LIN {X 99.483,Y -60.000,Z -86.142,A -90.000,B 90.000,C 0.000} C_DIS
LIN {X 99.483,Y -29.308,Z -86.142,A -90.000,B 90.000,C 0.000} C_DIS
LIN {X 99.474,Y -29.310,Z -86.271,A -90.000,B 90.000,C 0.000} C_DIS
LIN {X 99.431,Y -29.338,Z -86.823,A -90.000,B 90.000,C 0.000} C_DIS
LIN {X 99.416,Y -29.357,Z -87.009,A -90.000,B 90.000,C 0.000} C_DIS
LIN {X 99.411,Y -29.358,Z -87.066,A -90.000,B 90.000,C 0.000} C_DIS
LIN {X 99.408,Y -29.365,Z -87.238,A -90.000,B 90.000,C 0.000} C_DIS
LIN {X 99.404,Y -29.371,Z -87.535,A -90.000,B 90.000,C 0.000} C_DIS
LIN {X 99.396,Y -29.374,Z -87.741,A -90.000,B 90.000,C 0.000} C_DIS
LIN {X 99.366,Y -29.385,Z -88.382,A -90.000,B 90.000,C 0.000} C_DIS
LIN {X 99.349,Y -29.388,Z -88.757,A -90.000,B 90.000,C 0.000} C_DIS
LIN {X 99.326,Y -29.411,Z -90.340,A -90.000,B 90.000,C 0.000} C_DIS
LIN {X 99.319,Y -29.416,Z -90.874,A -90.000,B 90.000,C 0.000} C_DIS
LIN {X 99.295,Y -29.416,Z -91.496,A -90.000,B 90.000,C 0.000} C_DIS
LIN {X 99.271,Y -29.421,Z -92.100,A -90.000,B 90.000,C 0.000} C_DIS
LIN {X 99.242,Y -29.426,Z -92.749,A -90.000,B 90.000,C 0.000} C_DIS
LIN {X 99.174,Y -29.426,Z -93.750,A -90.000,B 90.000,C 0.000} C_DIS
LIN {X 99.148,Y -29.428,Z -94.121,A -90.000,B 90.000,C 0.000} C_DIS
LIN {X 99.143,Y -29.428,Z -94.158,A -90.000,B 90.000,C 0.000} C_DIS
LIN {X 99.082,Y -29.425,Z -94.592,A -90.000,B 90.000,C 0.000} C_DIS
LIN {X 98.973,Y -29.414,Z -95.189,A -90.000,B 90.000,C 0.000} C_DIS
LIN {X 98.893,Y -29.411,Z -95.613,A -90.000,B 90.000,C 0.000} C_DIS
LIN {X 98.843,Y -29.411,Z -95.835,A -90.000,B 90.000,C 0.000} C_DIS
LIN {X 98.623,Y -29.420,Z -96.806,A -90.000,B 90.000,C 0.000} C_DIS
LIN {X 98.597,Y -29.422,Z -96.941,A -90.000,B 90.000,C 0.000} C_DIS
LIN {X 98.549,Y -29.421,Z -97.133,A -90.000,B 90.000,C 0.000} C_DIS
LIN {X 98.489,Y -29.424,Z -97.369,A -90.000,B 90.000,C 0.000} C_DIS
LIN {X 98.242,Y -29.426,Z -98.215,A -90.000,B 90.000,C 0.000} C_DIS
LIN {X 98.196,Y -29.431,Z -98.439,A -90.000,B 90.000,C 0.000} C_DIS
LIN {X 98.116,Y -29.446,Z -98.815,A -90.000,B 90.000,C 0.000} C_DIS
LIN {X 98.030,Y -29.468,Z -99.250,A -90.000,B 90.000,C 0.000} C_DIS
LIN {X 97.907,Y -29.486,Z -99.897,A -90.000,B 90.000,C 0.000} C_DIS
LIN {X 97.776,Y -29.509,Z -100.630,A -90.000,B 90.000,C 0.000} C_DIS
LIN {X 97.672,Y -29.519,Z -101.231,A -90.000,B 90.000,C 0.000} C_DIS
LIN {X 97.614,Y -29.526,Z -101.574,A -90.000,B 90.000,C 0.000} C_DIS
LIN {X 97.555,Y -29.538,Z -101.977,A -90.000,B 90.000,C 0.000} C_DIS
LIN {X 97.524,Y -29.542,Z -102.200,A -90.000,B 90.000,C 0.000} C_DIS
LIN {X 97.389,Y -29.552,Z -103.092,A -90.000,B 90.000,C 0.000} C_DIS
LIN {X 97.380,Y -29.555,Z -103.178,A -90.000,B 90.000,C 0.000} C_DIS
LIN {X 97.349,Y -29.565,Z -103.442,A -90.000,B 90.000,C 0.000} C_DIS
LIN {X 97.261,Y -29.575,Z -104.227,A -90.000,B 90.000,C 0.000} C_DIS
LIN {X 97.256,Y -29.586,Z -104.403,A -90.000,B 90.000,C 0.000} C_DIS
LIN {X 97.253,Y -29.592,Z -104.507,A -90.000,B 90.000,C 0.000} C_DIS
LIN {X 97.252,Y -29.598,Z -105.008,A -90.000,B 90.000,C 0.000} C_DIS
LIN {X 97.255,Y -29.601,Z -105.049,A -90.000,B 90.000,C 0.000} C_DIS
LIN {X 97.332,Y -29.605,Z -105.759,A -90.000,B 90.000,C 0.000} C_DIS
LIN {X 97.345,Y -29.602,Z -105.867,A -90.000,B 90.000,C 0.000} C_DIS
LIN {X 97.415,Y -29.603,Z -106.286,A -90.000,B 90.000,C 0.000} C_DIS
LIN {X 97.518,Y -29.607,Z -106.935,A -90.000,B 90.000,C 0.000} C_DIS
LIN {X 97.664,Y -29.611,Z -107.964,A -90.000,B 90.000,C 0.000} C_DIS
LIN {X 97.689,Y -29.614,Z -108.147,A -90.000,B 90.000,C 0.000} C_DIS
LIN {X 97.799,Y -29.623,Z -109.641,A -90.000,B 90.000,C 0.000} C_DIS
LIN {X 97.823,Y -29.623,Z -110.079,A -90.000,B 90.000,C 0.000} C_DIS
LIN {X 97.850,Y -29.627,Z -110.772,A -90.000,B 90.000,C 0.000} C_DIS
LIN {X 97.887,Y -29.631,Z -111.828,A -90.000,B 90.000,C 0.000} C_DIS
LIN {X 97.974,Y -29.650,Z -115.821,A -90.000,B 90.000,C 0.000} C_DIS
LIN {X 98.033,Y -29.661,Z -117.860,A -90.000,B 90.000,C 0.000} C_DIS
LIN {X 98.103,Y -29.670,Z -120.291,A -90.000,B 90.000,C 0.000} C_DIS
LIN {X 98.151,Y -29.676,Z -122.571,A -90.000,B 90.000,C 0.000} C_DIS
LIN {X 98.155,Y -29.681,Z -124.129,A -90.000,B 90.000,C 0.000} C_DIS
LIN {X 98.155,Y -29.682,Z -124.889,A -90.000,B 90.000,C 0.000} C_DIS
LIN {X 98.140,Y -29.682,Z -125.406,A -90.000,B 90.000,C 0.000} C_DIS
LIN {X 98.088,Y -29.690,Z -127.201,A -90.000,B 90.000,C 0.000} C_DIS
LIN {X 98.040,Y -29.694,Z -128.030,A -90.000,B 90.000,C 0.000} C_DIS
LIN {X 97.964,Y -29.700,Z -129.451,A -90.000,B 90.000,C 0.000} C_DIS
LIN {X 97.879,Y -29.705,Z -130.608,A -90.000,B 90.000,C 0.000} C_DIS
LIN {X 97.791,Y -29.710,Z -131.863,A -90.000,B 90.000,C 0.000} C_DIS
LIN {X 97.673,Y -29.714,Z -133.353,A -90.000,B 90.000,C 0.000} C_DIS
LIN {X 97.534,Y -29.719,Z -135.178,A -90.000,B 90.000,C 0.000} C_DIS
LIN {X 97.341,Y -29.723,Z -137.704,A -90.000,B 90.000,C 0.000} C_DIS
LIN {X 97.283,Y -29.724,Z -138.417,A -90.000,B 90.000,C 0.000} C_DIS
LIN {X 97.044,Y -29.726,Z -141.288,A -90.000,B 90.000,C 0.000} C_DIS
LIN {X 97.013,Y -29.725,Z -141.637,A -90.000,B 90.000,C 0.000} C_DIS
LIN {X 96.932,Y -29.726,Z -142.492,A -90.000,B 90.000,C 0.000} C_DIS
LIN {X 96.735,Y -29.726,Z -144.533,A -90.000,B 90.000,C 0.000} C_DIS
LIN {X 96.664,Y -29.726,Z -145.241,A -90.000,B 90.000,C 0.000} C_DIS
LIN {X 96.504,Y -29.729,Z -146.660,A -90.000,B 90.000,C 0.000} C_DIS
LIN {X 96.220,Y -29.731,Z -149.069,A -90.000,B 90.000,C 0.000} C_DIS
LIN {X 96.032,Y -29.735,Z -150.385,A -90.000,B 90.000,C 0.000} C_DIS
LIN {X 95.981,Y -29.735,Z -150.733,A -90.000,B 90.000,C 0.000} C_DIS
LIN {X 95.686,Y -29.738,Z -152.718,A -90.000,B 90.000,C 0.000} C_DIS
LIN {X 95.484,Y -29.744,Z -153.901,A -90.000,B 90.000,C 0.000} C_DIS
LIN {X 95.283,Y -29.745,Z -155.034,A -90.000,B 90.000,C 0.000} C_DIS
LIN {X 95.055,Y -29.748,Z -156.296,A -90.000,B 90.000,C 0.000} C_DIS
LIN {X 94.789,Y -29.756,Z -157.638,A -90.000,B 90.000,C 0.000} C_DIS
LIN {X 94.604,Y -29.760,Z -158.553,A -90.000,B 90.000,C 0.000} C_DIS
LIN {X 94.410,Y -29.762,Z -159.484,A -90.000,B 90.000,C 0.000} C_DIS
LIN {X 94.217,Y -29.764,Z -160.395,A -90.000,B 90.000,C 0.000} C_DIS
LIN {X 93.802,Y -29.779,Z -162.241,A -90.000,B 90.000,C 0.000} C_DIS
LIN {X 93.711,Y -29.780,Z -162.635,A -90.000,B 90.000,C 0.000} C_DIS
LIN {X 93.376,Y -29.787,Z -164.032,A -90.000,B 90.000,C 0.000} C_DIS
LIN {X 92.902,Y -29.804,Z -165.942,A -90.000,B 90.000,C 0.000} C_DIS
LIN {X 92.850,Y -29.804,Z -166.143,A -90.000,B 90.000,C 0.000} C_DIS
LIN {X 92.491,Y -29.812,Z -167.498,A -90.000,B 90.000,C 0.000} C_DIS
LIN {X 91.956,Y -29.832,Z -169.511,A -90.000,B 90.000,C 0.000} C_DIS
LIN {X 91.869,Y -29.832,Z -169.825,A -90.000,B 90.000,C 0.000} C_DIS
LIN {X 91.493,Y -29.840,Z -171.143,A -90.000,B 90.000,C 0.000} C_DIS
LIN {X 90.972,Y -29.862,Z -173.009,A -90.000,B 90.000,C 0.000} C_DIS
LIN {X 90.878,Y -29.863,Z -173.340,A -90.000,B 90.000,C 0.000} C_DIS
LIN {X 90.675,Y -29.872,Z -174.031,A -90.000,B 90.000,C 0.000} C_DIS
LIN {X 90.451,Y -29.877,Z -174.778,A -90.000,B 90.000,C 0.000} C_DIS
LIN {X 89.905,Y -29.900,Z -176.678,A -90.000,B 90.000,C 0.000} C_DIS
LIN {X 89.709,Y -29.912,Z -177.349,A -90.000,B 90.000,C 0.000} C_DIS
LIN {X 89.267,Y -29.923,Z -178.782,A -90.000,B 90.000,C 0.000} C_DIS
LIN {X 89.182,Y -29.928,Z -179.064,A -90.000,B 90.000,C 0.000} C_DIS
LIN {X 88.588,Y -29.956,Z -181.124,A -90.000,B 90.000,C 0.000} C_DIS
LIN {X 88.497,Y -29.957,Z -181.422,A -90.000,B 90.000,C 0.000} C_DIS
LIN {X 88.343,Y -29.970,Z -181.945,A -90.000,B 90.000,C 0.000} C_DIS
LIN {X 87.960,Y -29.993,Z -183.282,A -90.000,B 90.000,C 0.000} C_DIS
LIN {X 87.916,Y -29.999,Z -183.447,A -90.000,B 90.000,C 0.000} C_DIS
LIN {X 87.747,Y -30.012,Z -184.045,A -90.000,B 90.000,C 0.000} C_DIS
LIN {X 87.596,Y -30.027,Z -184.565,A -90.000,B 90.000,C 0.000} C_DIS
LIN {X 87.334,Y -30.047,Z -185.497,A -90.000,B 90.000,C 0.000} C_DIS
LIN {X 87.245,Y -30.061,Z -185.833,A -90.000,B 90.000,C 0.000} C_DIS
LIN {X 87.002,Y -30.086,Z -186.710,A -90.000,B 90.000,C 0.000} C_DIS
LIN {X 86.920,Y -30.096,Z -186.998,A -90.000,B 90.000,C 0.000} C_DIS
LIN {X 86.846,Y -30.103,Z -187.267,A -90.000,B 90.000,C 0.000} C_DIS
LIN {X 86.560,Y -30.159,Z -188.385,A -90.000,B 90.000,C 0.000} C_DIS
LIN {X 86.479,Y -30.172,Z -188.756,A -90.000,B 90.000,C 0.000} C_DIS
LIN {X 86.380,Y -30.187,Z -189.229,A -90.000,B 90.000,C 0.000} C_DIS
LIN {X 86.321,Y -30.198,Z -189.479,A -90.000,B 90.000,C 0.000} C_DIS
LIN {X 86.005,Y -30.231,Z -190.710,A -90.000,B 90.000,C 0.000} C_DIS
LIN {X 85.884,Y -30.254,Z -191.208,A -90.000,B 90.000,C 0.000} C_DIS
LIN {X 85.716,Y -30.279,Z -192.000,A -90.000,B 90.000,C 0.000} C_DIS
LIN {X 85.660,Y -30.289,Z -192.248,A -90.000,B 90.000,C 0.000} C_DIS
LIN {X 85.508,Y -30.308,Z -192.903,A -90.000,B 90.000,C 0.000} C_DIS
LIN {X 85.408,Y -30.319,Z -193.291,A -90.000,B 90.000,C 0.000} C_DIS
LIN {X 85.234,Y -30.347,Z -193.986,A -90.000,B 90.000,C 0.000} C_DIS
LIN {X 84.749,Y -30.413,Z -196.124,A -90.000,B 90.000,C 0.000} C_DIS
LIN {X 84.616,Y -30.429,Z -196.622,A -90.000,B 90.000,C 0.000} C_DIS
LIN {X 84.518,Y -30.446,Z -196.992,A -90.000,B 90.000,C 0.000} C_DIS
LIN {X 83.870,Y -30.530,Z -199.637,A -90.000,B 90.000,C 0.000} C_DIS
LIN {X 83.793,Y -30.538,Z -199.989,A -90.000,B 90.000,C 0.000} C_DIS
LIN {X 83.689,Y -30.546,Z -200.503,A -90.000,B 90.000,C 0.000} C_DIS
LIN {X 83.582,Y -30.556,Z -201.000,A -90.000,B 90.000,C 0.000} C_DIS
LIN {X 83.401,Y -30.566,Z -201.831,A -90.000,B 90.000,C 0.000} C_DIS
LIN {X 83.009,Y -30.597,Z -203.446,A -90.000,B 90.000,C 0.000} C_DIS
LIN {X 82.848,Y -30.611,Z -204.109,A -90.000,B 90.000,C 0.000} C_DIS
LIN {X 82.270,Y -30.648,Z -206.753,A -90.000,B 90.000,C 0.000} C_DIS
LIN {X 82.070,Y -30.653,Z -207.647,A -90.000,B 90.000,C 0.000} C_DIS
LIN {X 81.809,Y -30.672,Z -208.669,A -90.000,B 90.000,C 0.000} C_DIS
LIN {X 81.175,Y -30.709,Z -211.483,A -90.000,B 90.000,C 0.000} C_DIS
LIN {X 80.817,Y -30.722,Z -213.179,A -90.000,B 90.000,C 0.000} C_DIS
LIN {X 80.751,Y -30.722,Z -213.489,A -90.000,B 90.000,C 0.000} C_DIS
LIN {X 80.529,Y -30.706,Z -214.656,A -90.000,B 90.000,C 0.000} C_DIS
LIN {X 80.221,Y -30.686,Z -216.247,A -90.000,B 90.000,C 0.000} C_DIS
LIN {X 80.023,Y -30.682,Z -217.167,A -90.000,B 90.000,C 0.000} C_DIS
LIN {X 79.724,Y -30.689,Z -218.572,A -90.000,B 90.000,C 0.000} C_DIS
LIN {X 79.476,Y -30.690,Z -219.646,A -90.000,B 90.000,C 0.000} C_DIS
LIN {X 79.237,Y -30.652,Z -221.129,A -90.000,B 90.000,C 0.000} C_DIS
LIN {X 79.196,Y -30.649,Z -221.387,A -90.000,B 90.000,C 0.000} C_DIS
LIN {X 79.079,Y -30.640,Z -222.126,A -90.000,B 90.000,C 0.000} C_DIS
LIN {X 78.730,Y -30.641,Z -223.935,A -90.000,B 90.000,C 0.000} C_DIS
LIN {X 78.437,Y -30.631,Z -225.264,A -90.000,B 90.000,C 0.000} C_DIS
LIN {X 77.635,Y -30.671,Z -228.599,A -90.000,B 90.000,C 0.000} C_DIS
LIN {X 77.465,Y -30.671,Z -229.435,A -90.000,B 90.000,C 0.000} C_DIS
LIN {X 77.439,Y -30.669,Z -229.557,A -90.000,B 90.000,C 0.000} C_DIS
LIN {X 77.335,Y -30.672,Z -229.945,A -90.000,B 90.000,C 0.000} C_DIS
LIN {X 76.486,Y -30.675,Z -233.044,A -90.000,B 90.000,C 0.000} C_DIS
LIN {X 76.190,Y -30.661,Z -234.259,A -90.000,B 90.000,C 0.000} C_DIS
LIN {X 75.999,Y -30.647,Z -235.042,A -90.000,B 90.000,C 0.000} C_DIS
LIN {X 75.922,Y -30.644,Z -235.352,A -90.000,B 90.000,C 0.000} C_DIS
LIN {X 75.147,Y -30.631,Z -237.779,A -90.000,B 90.000,C 0.000} C_DIS
LIN {X 74.482,Y -30.600,Z -240.000,A -90.000,B 90.000,C 0.000} C_DIS
LIN {X 74.079,Y -30.591,Z -241.357,A -90.000,B 90.000,C 0.000} C_DIS
LIN {X 74.045,Y -30.588,Z -241.457,A -90.000,B 90.000,C 0.000} C_DIS
LIN {X 73.948,Y -30.585,Z -241.722,A -90.000,B 90.000,C 0.000} C_DIS
LIN {X 73.618,Y -30.580,Z -242.599,A -90.000,B 90.000,C 0.000} C_DIS
LIN {X 73.258,Y -30.572,Z -243.561,A -90.000,B 90.000,C 0.000} C_DIS
LIN {X 73.258,Y -60.000,Z -243.561,A -90.000,B 90.000,C 0.000} C_DIS
LIN {X 87.811,Y -60.000,Z -190.830,A -90.000,B 90.000,C 0.000} C_DIS
LIN {X 87.811,Y -29.308,Z -190.830,A -90.000,B 90.000,C 0.000} C_DIS
LIN {X 87.630,Y -29.365,Z -191.611,A -90.000,B 90.000,C 0.000} C_DIS
LIN {X 87.472,Y -29.410,Z -192.399,A -90.000,B 90.000,C 0.000} C_DIS
LIN {X 87.379,Y -29.436,Z -192.833,A -90.000,B 90.000,C 0.000} C_DIS
LIN {X 87.253,Y -29.462,Z -193.396,A -90.000,B 90.000,C 0.000} C_DIS
LIN {X 87.008,Y -29.527,Z -194.411,A -90.000,B 90.000,C 0.000} C_DIS
LIN {X 86.652,Y -29.613,Z -196.049,A -90.000,B 90.000,C 0.000} C_DIS
LIN {X 86.522,Y -29.635,Z -196.625,A -90.000,B 90.000,C 0.000} C_DIS
LIN {X 86.308,Y -29.679,Z -197.452,A -90.000,B 90.000,C 0.000} C_DIS
LIN {X 85.755,Y -29.786,Z -199.765,A -90.000,B 90.000,C 0.000} C_DIS
LIN {X 85.678,Y -29.796,Z -200.077,A -90.000,B 90.000,C 0.000} C_DIS
LIN {X 85.613,Y -29.801,Z -200.371,A -90.000,B 90.000,C 0.000} C_DIS
LIN {X 85.508,Y -29.808,Z -200.885,A -90.000,B 90.000,C 0.000} C_DIS
LIN {X 85.216,Y -29.830,Z -202.235,A -90.000,B 90.000,C 0.000} C_DIS
LIN {X 85.032,Y -29.851,Z -203.007,A -90.000,B 90.000,C 0.000} C_DIS
LIN {X 84.825,Y -29.877,Z -203.874,A -90.000,B 90.000,C 0.000} C_DIS
LIN {X 84.669,Y -29.889,Z -204.517,A -90.000,B 90.000,C 0.000} C_DIS
LIN {X 84.163,Y -29.908,Z -206.801,A -90.000,B 90.000,C 0.000} C_DIS
LIN {X 83.886,Y -29.924,Z -208.063,A -90.000,B 90.000,C 0.000} C_DIS
LIN {X 83.804,Y -29.933,Z -208.389,A -90.000,B 90.000,C 0.000} C_DIS
LIN {X 83.625,Y -29.945,Z -209.087,A -90.000,B 90.000,C 0.000} C_DIS
LIN {X 83.398,Y -29.950,Z -210.078,A -90.000,B 90.000,C 0.000} C_DIS
LIN {X 82.992,Y -29.969,Z -211.871,A -90.000,B 90.000,C 0.000} C_DIS
LIN {X 82.675,Y -29.978,Z -213.369,A -90.000,B 90.000,C 0.000} C_DIS
LIN {X 82.568,Y -29.977,Z -213.866,A -90.000,B 90.000,C 0.000} C_DIS
LIN {X 82.504,Y -29.972,Z -214.208,A -90.000,B 90.000,C 0.000} C_DIS
LIN {X 82.241,Y -29.966,Z -215.607,A -90.000,B 90.000,C 0.000} C_DIS
LIN {X 82.044,Y -29.961,Z -216.636,A -90.000,B 90.000,C 0.000} C_DIS
LIN {X 81.886,Y -29.962,Z -217.380,A -90.000,B 90.000,C 0.000} C_DIS
LIN {X 81.546,Y -29.965,Z -218.964,A -90.000,B 90.000,C 0.000} C_DIS
LIN {X 81.487,Y -29.967,Z -219.226,A -90.000,B 90.000,C 0.000} C_DIS
LIN {X 81.310,Y -29.971,Z -219.998,A -90.000,B 90.000,C 0.000} C_DIS
LIN {X 81.177,Y -29.942,Z -220.804,A -90.000,B 90.000,C 0.000} C_DIS
LIN {X 80.910,Y -29.887,Z -222.408,A -90.000,B 90.000,C 0.000} C_DIS
LIN {X 80.805,Y -29.877,Z -222.936,A -90.000,B 90.000,C 0.000} C_DIS
LIN {X 80.572,Y -29.866,Z -224.118,A -90.000,B 90.000,C 0.000} C_DIS
LIN {X 80.538,Y -29.862,Z -224.285,A -90.000,B 90.000,C 0.000} C_DIS
LIN {X 80.234,Y -29.843,Z -225.653,A -90.000,B 90.000,C 0.000} C_DIS
LIN {X 79.868,Y -29.839,Z -227.137,A -90.000,B 90.000,C 0.000} C_DIS
LIN {X 79.414,Y -29.850,Z -229.007,A -90.000,B 90.000,C 0.000} C_DIS
LIN {X 79.282,Y -29.844,Z -229.639,A -90.000,B 90.000,C 0.000} C_DIS
LIN {X 79.220,Y -29.838,Z -229.924,A -90.000,B 90.000,C 0.000} C_DIS
LIN {X 79.194,Y -29.836,Z -230.032,A -90.000,B 90.000,C 0.000} C_DIS
LIN {X 78.636,Y -29.828,Z -232.056,A -90.000,B 90.000,C 0.000} C_DIS
LIN {X 78.254,Y -29.835,Z -233.462,A -90.000,B 90.000,C 0.000} C_DIS
LIN {X 77.714,Y -29.816,Z -235.688,A -90.000,B 90.000,C 0.000} C_DIS
LIN {X 77.690,Y -29.813,Z -235.781,A -90.000,B 90.000,C 0.000} C_DIS
LIN {X 77.655,Y -29.810,Z -235.901,A -90.000,B 90.000,C 0.000} C_DIS
LIN {X 77.381,Y -29.806,Z -236.760,A -90.000,B 90.000,C 0.000} C_DIS
LIN {X 76.897,Y -29.807,Z -238.290,A -90.000,B 90.000,C 0.000} C_DIS
LIN {X 75.883,Y -29.783,Z -241.710,A -90.000,B 90.000,C 0.000} C_DIS
LIN {X 75.833,Y -29.778,Z -241.871,A -90.000,B 90.000,C 0.000} C_DIS
LIN {X 75.781,Y -29.775,Z -242.026,A -90.000,B 90.000,C 0.000} C_DIS
LIN {X 75.660,Y -29.772,Z -242.361,A -90.000,B 90.000,C 0.000} C_DIS
LIN {X 75.382,Y -29.771,Z -243.105,A -90.000,B 90.000,C 0.000} C_DIS
LIN {X 75.211,Y -29.767,Z -243.561,A -90.000,B 90.000,C 0.000} C_DIS
LIN {X 75.211,Y -60.000,Z -243.561,A -90.000,B 90.000,C 0.000} C_DIS
LIN {X -101.340,Y -60.000,Z -243.561,A -90.000,B 90.000,C 0.000} C_DIS
LIN {X -101.340,Y -30.001,Z -243.561,A -90.000,B 90.000,C 0.000} C_DIS
LIN {X -101.281,Y -29.939,Z -243.470,A -90.000,B 90.000,C 0.000} C_DIS
LIN {X -101.216,Y -29.882,Z -243.379,A -90.000,B 90.000,C 0.000} C_DIS
LIN {X -101.156,Y -29.837,Z -243.300,A -90.000,B 90.000,C 0.000} C_DIS
LIN {X -100.984,Y -29.743,Z -243.101,A -90.000,B 90.000,C 0.000} C_DIS
LIN {X -100.897,Y -29.711,Z -243.012,A -90.000,B 90.000,C 0.000} C_DIS
LIN {X -100.794,Y -29.682,Z -242.913,A -90.000,B 90.000,C 0.000} C_DIS
LIN {X -100.571,Y -29.651,Z -242.724,A -90.000,B 90.000,C 0.000} C_DIS
LIN {X -100.388,Y -29.648,Z -242.588,A -90.000,B 90.000,C 0.000} C_DIS
LIN {X -100.243,Y -29.644,Z -242.486,A -90.000,B 90.000,C 0.000} C_DIS
LIN {X -99.888,Y -29.641,Z -242.242,A -90.000,B 90.000,C 0.000} C_DIS
LIN {X -97.039,Y -29.629,Z -240.290,A -90.000,B 90.000,C 0.000} C_DIS
LIN {X -94.571,Y -29.636,Z -238.566,A -90.000,B 90.000,C 0.000} C_DIS
LIN {X -92.711,Y -29.631,Z -237.259,A -90.000,B 90.000,C 0.000} C_DIS
LIN {X -92.062,Y -29.616,Z -236.829,A -90.000,B 90.000,C 0.000} C_DIS
LIN {X -91.234,Y -29.615,Z -236.292,A -90.000,B 90.000,C 0.000} C_DIS
LIN {X -87.893,Y -29.631,Z -234.084,A -90.000,B 90.000,C 0.000} C_DIS
LIN {X -84.347,Y -29.626,Z -231.735,A -90.000,B 90.000,C 0.000} C_DIS
LIN {X -83.919,Y -29.620,Z -231.462,A -90.000,B 90.000,C 0.000} C_DIS
LIN {X -81.041,Y -29.630,Z -229.677,A -90.000,B 90.000,C 0.000} C_DIS
LIN {X -77.308,Y -29.632,Z -227.354,A -90.000,B 90.000,C 0.000} C_DIS
LIN {X -75.762,Y -29.629,Z -226.401,A -90.000,B 90.000,C 0.000} C_DIS
LIN {X -75.399,Y -29.624,Z -226.188,A -90.000,B 90.000,C 0.000} C_DIS
LIN {X -74.549,Y -29.623,Z -225.699,A -90.000,B 90.000,C 0.000} C_DIS
LIN {X -72.247,Y -29.625,Z -224.377,A -90.000,B 90.000,C 0.000} C_DIS
LIN {X -68.413,Y -29.640,Z -222.185,A -90.000,B 90.000,C 0.000} C_DIS
LIN {X -67.099,Y -29.645,Z -221.436,A -90.000,B 90.000,C 0.000} C_DIS
LIN {X -66.651,Y -29.644,Z -221.189,A -90.000,B 90.000,C 0.000} C_DIS
LIN {X -65.033,Y -29.654,Z -220.309,A -90.000,B 90.000,C 0.000} C_DIS
LIN {X -60.798,Y -29.693,Z -218.013,A -90.000,B 90.000,C 0.000} C_DIS
LIN {X -58.582,Y -29.708,Z -216.827,A -90.000,B 90.000,C 0.000} C_DIS
LIN {X -58.020,Y -29.710,Z -216.529,A -90.000,B 90.000,C 0.000} C_DIS
LIN {X -54.719,Y -29.743,Z -214.797,A -90.000,B 90.000,C 0.000} C_DIS
LIN {X -53.441,Y -29.750,Z -214.136,A -90.000,B 90.000,C 0.000} C_DIS
LIN {X -50.611,Y -29.771,Z -212.676,A -90.000,B 90.000,C 0.000} C_DIS
LIN {X -49.077,Y -29.785,Z -211.879,A -90.000,B 90.000,C 0.000} C_DIS
LIN {X -48.337,Y -29.788,Z -211.498,A -90.000,B 90.000,C 0.000} C_DIS
LIN {X -44.173,Y -29.810,Z -209.360,A -90.000,B 90.000,C 0.000} C_DIS
LIN {X -43.553,Y -29.812,Z -209.043,A -90.000,B 90.000,C 0.000} C_DIS
LIN {X -43.086,Y -29.818,Z -208.799,A -90.000,B 90.000,C 0.000} C_DIS
LIN {X -40.938,Y -29.823,Z -207.653,A -90.000,B 90.000,C 0.000} C_DIS
LIN {X -38.034,Y -29.831,Z -206.106,A -90.000,B 90.000,C 0.000} C_DIS
LIN {X -37.736,Y -29.835,Z -205.943,A -90.000,B 90.000,C 0.000} C_DIS
LIN {X -36.183,Y -29.830,Z -205.071,A -90.000,B 90.000,C 0.000} C_DIS
LIN {X -33.862,Y -29.831,Z -203.772,A -90.000,B 90.000,C 0.000} C_DIS
LIN {X -33.306,Y -29.832,Z -203.456,A -90.000,B 90.000,C 0.000} C_DIS
LIN {X -33.015,Y -29.836,Z -203.285,A -90.000,B 90.000,C 0.000} C_DIS
LIN {X -30.370,Y -29.831,Z -201.691,A -90.000,B 90.000,C 0.000} C_DIS
LIN {X -29.687,Y -29.833,Z -201.273,A -90.000,B 90.000,C 0.000} C_DIS
LIN {X -29.246,Y -29.832,Z -201.001,A -90.000,B 90.000,C 0.000} C_DIS
LIN {X -28.989,Y -29.836,Z -200.838,A -90.000,B 90.000,C 0.000} C_DIS
LIN {X -27.015,Y -29.833,Z -199.551,A -90.000,B 90.000,C 0.000} C_DIS
LIN {X -26.253,Y -29.834,Z -199.046,A -90.000,B 90.000,C 0.000} C_DIS
LIN {X -25.666,Y -29.833,Z -198.657,A -90.000,B 90.000,C 0.000} C_DIS
LIN {X -25.567,Y -29.834,Z -198.590,A -90.000,B 90.000,C 0.000} C_DIS
LIN {X -24.143,Y -29.832,Z -197.587,A -90.000,B 90.000,C 0.000} C_DIS
LIN {X -22.628,Y -29.834,Z -196.527,A -90.000,B 90.000,C 0.000} C_DIS
LIN {X -22.375,Y -29.839,Z -196.343,A -90.000,B 90.000,C 0.000} C_DIS
LIN {X -20.722,Y -29.839,Z -195.100,A -90.000,B 90.000,C 0.000} C_DIS
LIN {X -19.359,Y -29.845,Z -194.074,A -90.000,B 90.000,C 0.000} C_DIS
LIN {X -19.097,Y -29.850,Z -193.870,A -90.000,B 90.000,C 0.000} C_DIS
LIN {X -17.597,Y -29.853,Z -192.672,A -90.000,B 90.000,C 0.000} C_DIS
LIN {X -16.118,Y -29.863,Z -191.477,A -90.000,B 90.000,C 0.000} C_DIS
LIN {X -15.815,Y -29.869,Z -191.226,A -90.000,B 90.000,C 0.000} C_DIS
LIN {X -14.190,Y -29.877,Z -189.854,A -90.000,B 90.000,C 0.000} C_DIS
LIN {X -13.835,Y -29.881,Z -189.550,A -90.000,B 90.000,C 0.000} C_DIS
LIN {X -13.069,Y -29.889,Z -188.890,A -90.000,B 90.000,C 0.000} C_DIS
LIN {X -12.496,Y -29.905,Z -188.382,A -90.000,B 90.000,C 0.000} C_DIS
LIN {X -11.099,Y -29.922,Z -187.114,A -90.000,B 90.000,C 0.000} C_DIS
LIN {X -10.495,Y -29.934,Z -186.572,A -90.000,B 90.000,C 0.000} C_DIS
LIN {X -9.651,Y -29.940,Z -185.828,A -90.000,B 90.000,C 0.000} C_DIS
LIN {X -9.103,Y -29.961,Z -185.324,A -90.000,B 90.000,C 0.000} C_DIS
LIN {X -7.768,Y -29.980,Z -184.048,A -90.000,B 90.000,C 0.000} C_DIS
LIN {X -6.999,Y -30.000,Z -183.326,A -90.000,B 90.000,C 0.000} C_DIS
LIN {X -6.189,Y -30.009,Z -182.580,A -90.000,B 90.000,C 0.000} C_DIS
LIN {X -5.899,Y -30.029,Z -182.294,A -90.000,B 90.000,C 0.000} C_DIS
LIN {X -5.606,Y -30.043,Z -182.013,A -90.000,B 90.000,C 0.000} C_DIS
LIN {X -3.248,Y -30.090,Z -179.616,A -90.000,B 90.000,C 0.000} C_DIS
LIN {X -2.903,Y -30.103,Z -179.275,A -90.000,B 90.000,C 0.000} C_DIS
LIN {X -2.326,Y -30.153,Z -178.675,A -90.000,B 90.000,C 0.000} C_DIS
LIN {X -1.394,Y -30.196,Z -177.629,A -90.000,B 90.000,C 0.000} C_DIS
LIN {X -0.006,Y -30.236,Z -176.096,A -90.000,B 90.000,C 0.000} C_DIS
LIN {X 0.206,Y -30.252,Z -175.855,A -90.000,B 90.000,C 0.000} C_DIS
LIN {X 0.398,Y -30.269,Z -175.644,A -90.000,B 90.000,C 0.000} C_DIS
LIN {X 0.477,Y -30.275,Z -175.553,A -90.000,B 90.000,C 0.000} C_DIS
LIN {X 0.513,Y -30.276,Z -175.507,A -90.000,B 90.000,C 0.000} C_DIS
LIN {X 1.881,Y -30.370,Z -173.737,A -90.000,B 90.000,C 0.000} C_DIS
LIN {X 2.269,Y -30.382,Z -173.186,A -90.000,B 90.000,C 0.000} C_DIS
LIN {X 2.623,Y -30.420,Z -172.664,A -90.000,B 90.000,C 0.000} C_DIS
LIN {X 2.752,Y -30.430,Z -172.460,A -90.000,B 90.000,C 0.000} C_DIS
LIN {X 3.183,Y -30.443,Z -171.680,A -90.000,B 90.000,C 0.000} C_DIS
LIN {X 3.433,Y -30.453,Z -171.240,A -90.000,B 90.000,C 0.000} C_DIS
LIN {X 3.831,Y -30.494,Z -170.516,A -90.000,B 90.000,C 0.000} C_DIS
LIN {X 4.063,Y -30.505,Z -170.017,A -90.000,B 90.000,C 0.000} C_DIS
LIN {X 4.092,Y -30.504,Z -169.943,A -90.000,B 90.000,C 0.000} C_DIS
LIN {X 4.243,Y -30.514,Z -169.540,A -90.000,B 90.000,C 0.000} C_DIS
LIN {X 4.327,Y -30.528,Z -169.306,A -90.000,B 90.000,C 0.000} C_DIS
LIN {X 4.479,Y -30.541,Z -168.749,A -90.000,B 90.000,C 0.000} C_DIS
LIN {X 4.578,Y -30.549,Z -168.398,A -90.000,B 90.000,C 0.000} C_DIS
LIN {X 4.757,Y -30.557,Z -167.779,A -90.000,B 90.000,C 0.000} C_DIS
LIN {X 4.783,Y -30.558,Z -167.696,A -90.000,B 90.000,C 0.000} C_DIS
LIN {X 4.861,Y -30.547,Z -167.303,A -90.000,B 90.000,C 0.000} C_DIS
LIN {X 4.927,Y -30.551,Z -166.945,A -90.000,B 90.000,C 0.000} C_DIS
LIN {X 4.955,Y -30.544,Z -166.651,A -90.000,B 90.000,C 0.000} C_DIS
LIN {X 4.956,Y -30.525,Z -166.356,A -90.000,B 90.000,C 0.000} C_DIS
LIN {X 4.959,Y -30.520,Z -166.265,A -90.000,B 90.000,C 0.000} C_DIS
LIN {X 4.966,Y -30.514,Z -165.878,A -90.000,B 90.000,C 0.000} C_DIS
LIN {X 4.963,Y -30.534,Z -165.505,A -90.000,B 90.000,C 0.000} C_DIS
LIN {X 4.978,Y -30.569,Z -164.942,A -90.000,B 90.000,C 0.000} C_DIS
LIN {X 4.935,Y -30.559,Z -164.645,A -90.000,B 90.000,C 0.000} C_DIS
LIN {X 4.797,Y -30.506,Z -163.606,A -90.000,B 90.000,C 0.000} C_DIS
LIN {X 4.450,Y -30.395,Z -163.003,A -90.000,B 90.000,C 0.000} C_DIS
LIN {X 4.140,Y -30.395,Z -162.548,A -90.000,B 90.000,C 0.000} C_DIS
LIN {X 3.659,Y -30.374,Z -161.821,A -90.000,B 90.000,C 0.000} C_DIS
LIN {X 3.582,Y -30.372,Z -161.703,A -90.000,B 90.000,C 0.000} C_DIS
LIN {X 3.144,Y -30.291,Z -161.267,A -90.000,B 90.000,C 0.000} C_DIS
LIN {X 2.852,Y -30.237,Z -160.973,A -90.000,B 90.000,C 0.000} C_DIS
LIN {X 2.821,Y -30.230,Z -160.941,A -90.000,B 90.000,C 0.000} C_DIS
LIN {X 2.556,Y -30.224,Z -160.707,A -90.000,B 90.000,C 0.000} C_DIS
LIN {X 1.968,Y -30.205,Z -160.173,A -90.000,B 90.000,C 0.000} C_DIS
LIN {X 1.376,Y -30.121,Z -159.761,A -90.000,B 90.000,C 0.000} C_DIS
LIN {X 0.749,Y -30.021,Z -159.300,A -90.000,B 90.000,C 0.000} C_DIS
LIN {X -0.029,Y -29.995,Z -158.816,A -90.000,B 90.000,C 0.000} C_DIS
LIN {X -0.158,Y -29.992,Z -158.731,A -90.000,B 90.000,C 0.000} C_DIS
LIN {X -0.255,Y -29.988,Z -158.667,A -90.000,B 90.000,C 0.000} C_DIS
LIN {X -0.451,Y -29.966,Z -158.554,A -90.000,B 90.000,C 0.000} C_DIS
LIN {X -0.931,Y -29.917,Z -158.274,A -90.000,B 90.000,C 0.000} C_DIS
LIN {X -1.598,Y -29.855,Z -157.874,A -90.000,B 90.000,C 0.000} C_DIS
LIN {X -2.685,Y -29.819,Z -157.286,A -90.000,B 90.000,C 0.000} C_DIS
LIN {X -2.985,Y -29.815,Z -157.113,A -90.000,B 90.000,C 0.000} C_DIS
LIN {X -3.332,Y -29.788,Z -156.935,A -90.000,B 90.000,C 0.000} C_DIS
LIN {X -3.746,Y -29.762,Z -156.717,A -90.000,B 90.000,C 0.000} C_DIS
LIN {X -4.215,Y -29.719,Z -156.449,A -90.000,B 90.000,C 0.000} C_DIS
LIN {X -4.775,Y -29.689,Z -156.156,A -90.000,B 90.000,C 0.000} C_DIS
LIN {X -5.829,Y -29.647,Z -155.619,A -90.000,B 90.000,C 0.000} C_DIS
LIN {X -6.235,Y -29.640,Z -155.407,A -90.000,B 90.000,C 0.000} C_DIS
LIN {X -6.910,Y -29.613,Z -155.062,A -90.000,B 90.000,C 0.000} C_DIS
LIN {X -8.240,Y -29.542,Z -154.339,A -90.000,B 90.000,C 0.000} C_DIS
LIN {X -8.931,Y -29.510,Z -153.959,A -90.000,B 90.000,C 0.000} C_DIS
LIN {X -9.555,Y -29.507,Z -153.628,A -90.000,B 90.000,C 0.000} C_DIS
LIN {X -9.642,Y -29.506,Z -153.580,A -90.000,B 90.000,C 0.000} C_DIS
LIN {X -11.121,Y -29.448,Z -152.682,A -90.000,B 90.000,C 0.000} C_DIS
LIN {X -11.642,Y -29.429,Z -152.363,A -90.000,B 90.000,C 0.000} C_DIS
LIN {X -12.443,Y -29.412,Z -151.908,A -90.000,B 90.000,C 0.000} C_DIS
LIN {X -12.828,Y -29.406,Z -151.665,A -90.000,B 90.000,C 0.000} C_DIS
LIN {X -14.136,Y -29.374,Z -150.774,A -90.000,B 90.000,C 0.000} C_DIS
LIN {X -14.875,Y -29.367,Z -150.307,A -90.000,B 90.000,C 0.000} C_DIS
LIN {X -15.778,Y -29.352,Z -149.737,A -90.000,B 90.000,C 0.000} C_DIS
LIN {X -16.098,Y -29.345,Z -149.510,A -90.000,B 90.000,C 0.000} C_DIS
LIN {X -16.203,Y -29.344,Z -149.434,A -90.000,B 90.000,C 0.000} C_DIS
LIN {X -16.596,Y -29.340,Z -149.140,A -90.000,B 90.000,C 0.000} C_DIS
LIN {X -18.379,Y -29.327,Z -147.883,A -90.000,B 90.000,C 0.000} C_DIS
LIN {X -19.359,Y -29.324,Z -147.231,A -90.000,B 90.000,C 0.000} C_DIS
LIN {X -19.862,Y -29.320,Z -146.844,A -90.000,B 90.000,C 0.000} C_DIS
LIN {X -20.614,Y -29.318,Z -146.256,A -90.000,B 90.000,C 0.000} C_DIS
LIN {X -23.023,Y -29.320,Z -144.446,A -90.000,B 90.000,C 0.000} C_DIS
LIN {X -23.262,Y -29.319,Z -144.261,A -90.000,B 90.000,C 0.000} C_DIS
LIN {X -23.388,Y -29.318,Z -144.160,A -90.000,B 90.000,C 0.000} C_DIS
LIN {X -24.392,Y -29.317,Z -143.290,A -90.000,B 90.000,C 0.000} C_DIS
LIN {X -25.941,Y -29.320,Z -141.982,A -90.000,B 90.000,C 0.000} C_DIS
LIN {X -26.769,Y -29.323,Z -141.273,A -90.000,B 90.000,C 0.000} C_DIS
LIN {X -26.925,Y -29.322,Z -141.125,A -90.000,B 90.000,C 0.000} C_DIS
LIN {X -27.122,Y -29.320,Z -140.936,A -90.000,B 90.000,C 0.000} C_DIS
LIN {X -28.391,Y -29.322,Z -139.639,A -90.000,B 90.000,C 0.000} C_DIS
LIN {X -29.230,Y -29.321,Z -138.774,A -90.000,B 90.000,C 0.000} C_DIS
LIN {X -30.310,Y -29.323,Z -137.693,A -90.000,B 90.000,C 0.000} C_DIS
LIN {X -30.624,Y -29.320,Z -137.321,A -90.000,B 90.000,C 0.000} C_DIS
LIN {X -30.894,Y -29.321,Z -136.990,A -90.000,B 90.000,C 0.000} C_DIS
LIN {X -32.972,Y -29.328,Z -134.427,A -90.000,B 90.000,C 0.000} C_DIS
LIN {X -33.191,Y -29.328,Z -134.153,A -90.000,B 90.000,C 0.000} C_DIS
LIN {X -33.263,Y -29.329,Z -134.064,A -90.000,B 90.000,C 0.000} C_DIS
LIN {X -33.544,Y -29.327,Z -133.662,A -90.000,B 90.000,C 0.000} C_DIS
LIN {X -35.140,Y -29.332,Z -131.218,A -90.000,B 90.000,C 0.000} C_DIS
LIN {X -35.789,Y -29.336,Z -130.229,A -90.000,B 90.000,C 0.000} C_DIS
LIN {X -35.985,Y -29.336,Z -129.875,A -90.000,B 90.000,C 0.000} C_DIS
LIN {X -36.025,Y -29.337,Z -129.804,A -90.000,B 90.000,C 0.000} C_DIS
LIN {X -36.701,Y -29.344,Z -128.522,A -90.000,B 90.000,C 0.000} C_DIS
LIN {X -37.699,Y -29.351,Z -126.570,A -90.000,B 90.000,C 0.000} C_DIS
LIN {X -37.813,Y -29.354,Z -126.346,A -90.000,B 90.000,C 0.000} C_DIS
LIN {X -38.010,Y -29.358,Z -125.889,A -90.000,B 90.000,C 0.000} C_DIS
LIN {X -38.906,Y -29.369,Z -123.626,A -90.000,B 90.000,C 0.000} C_DIS
LIN {X -39.262,Y -29.372,Z -122.689,A -90.000,B 90.000,C 0.000} C_DIS
LIN {X -39.399,Y -29.381,Z -122.321,A -90.000,B 90.000,C 0.000} C_DIS
LIN {X -39.551,Y -29.390,Z -121.868,A -90.000,B 90.000,C 0.000} C_DIS
LIN {X -39.562,Y -29.390,Z -121.827,A -90.000,B 90.000,C 0.000} C_DIS
LIN {X -39.892,Y -29.392,Z -120.578,A -90.000,B 90.000,C 0.000} C_DIS
LIN {X -40.370,Y -29.391,Z -118.778,A -90.000,B 90.000,C 0.000} C_DIS
LIN {X -40.456,Y -29.396,Z -118.449,A -90.000,B 90.000,C 0.000} C_DIS
LIN {X -40.716,Y -29.425,Z -117.427,A -90.000,B 90.000,C 0.000} C_DIS
LIN {X -40.853,Y -29.426,Z -116.619,A -90.000,B 90.000,C 0.000} C_DIS
LIN {X -41.233,Y -29.442,Z -114.619,A -90.000,B 90.000,C 0.000} C_DIS
LIN {X -41.316,Y -29.454,Z -114.177,A -90.000,B 90.000,C 0.000} C_DIS
LIN {X -41.365,Y -29.465,Z -113.913,A -90.000,B 90.000,C 0.000} C_DIS
LIN {X -41.495,Y -29.498,Z -113.309,A -90.000,B 90.000,C 0.000} C_DIS
LIN {X -41.702,Y -29.561,Z -112.445,A -90.000,B 90.000,C 0.000} C_DIS
LIN {X -41.726,Y -29.569,Z -112.342,A -90.000,B 90.000,C 0.000} C_DIS
LIN {X -41.770,Y -29.586,Z -112.182,A -90.000,B 90.000,C 0.000} C_DIS
LIN {X -41.973,Y -29.674,Z -111.533,A -90.000,B 90.000,C 0.000} C_DIS
LIN {X -42.096,Y -29.731,Z -111.135,A -90.000,B 90.000,C 0.000} C_DIS
LIN {X -42.185,Y -29.766,Z -110.857,A -90.000,B 90.000,C 0.000} C_DIS
LIN {X -42.308,Y -29.826,Z -110.542,A -90.000,B 90.000,C 0.000} C_DIS
LIN {X -42.449,Y -29.869,Z -110.221,A -90.000,B 90.000,C 0.000} C_DIS
LIN {X -42.648,Y -29.887,Z -109.836,A -90.000,B 90.000,C 0.000} C_DIS
LIN {X -42.794,Y -29.894,Z -109.541,A -90.000,B 90.000,C 0.000} C_DIS
LIN {X -42.817,Y -29.894,Z -109.496,A -90.000,B 90.000,C 0.000} C_DIS
LIN {X -42.920,Y -29.885,Z -109.317,A -90.000,B 90.000,C 0.000} C_DIS
LIN {X -43.524,Y -29.899,Z -108.384,A -90.000,B 90.000,C 0.000} C_DIS
LIN {X -43.607,Y -29.904,Z -108.251,A -90.000,B 90.000,C 0.000} C_DIS
LIN {X -44.099,Y -29.889,Z -107.528,A -90.000,B 90.000,C 0.000} C_DIS
LIN {X -44.437,Y -29.899,Z -107.064,A -90.000,B 90.000,C 0.000} C_DIS
LIN {X -44.775,Y -29.904,Z -106.594,A -90.000,B 90.000,C 0.000} C_DIS
LIN {X -45.307,Y -29.899,Z -105.877,A -90.000,B 90.000,C 0.000} C_DIS
LIN {X -45.897,Y -29.920,Z -105.123,A -90.000,B 90.000,C 0.000} C_DIS
LIN {X -46.438,Y -29.916,Z -104.465,A -90.000,B 90.000,C 0.000} C_DIS
LIN {X -46.828,Y -29.903,Z -103.975,A -90.000,B 90.000,C 0.000} C_DIS
LIN {X -47.346,Y -29.920,Z -103.326,A -90.000,B 90.000,C 0.000} C_DIS
LIN {X -47.964,Y -29.922,Z -102.580,A -90.000,B 90.000,C 0.000} C_DIS
LIN {X -48.540,Y -29.914,Z -101.867,A -90.000,B 90.000,C 0.000} C_DIS
LIN {X -48.782,Y -29.907,Z -101.562,A -90.000,B 90.000,C 0.000} C_DIS
LIN {X -48.953,Y -29.904,Z -101.342,A -90.000,B 90.000,C 0.000} C_DIS
LIN {X -49.469,Y -29.908,Z -100.657,A -90.000,B 90.000,C 0.000} C_DIS
LIN {X -50.281,Y -29.911,Z -99.575,A -90.000,B 90.000,C 0.000} C_DIS
LIN {X -50.697,Y -29.931,Z -99.016,A -90.000,B 90.000,C 0.000} C_DIS
LIN {X -50.882,Y -29.940,Z -98.766,A -90.000,B 90.000,C 0.000} C_DIS
LIN {X -51.320,Y -29.941,Z -98.148,A -90.000,B 90.000,C 0.000} C_DIS
LIN {X -51.561,Y -29.950,Z -97.796,A -90.000,B 90.000,C 0.000} C_DIS
LIN {X -52.278,Y -29.992,Z -96.764,A -90.000,B 90.000,C 0.000} C_DIS
LIN {X -52.883,Y -30.028,Z -95.890,A -90.000,B 90.000,C 0.000} C_DIS
LIN {X -53.078,Y -30.037,Z -95.604,A -90.000,B 90.000,C 0.000} C_DIS
LIN {X -53.478,Y -30.051,Z -95.008,A -90.000,B 90.000,C 0.000} C_DIS
LIN {X -53.991,Y -30.076,Z -94.229,A -90.000,B 90.000,C 0.000} C_DIS
LIN {X -54.307,Y -30.081,Z -93.732,A -90.000,B 90.000,C 0.000} C_DIS
LIN {X -55.041,Y -30.108,Z -92.537,A -90.000,B 90.000,C 0.000} C_DIS
LIN {X -55.186,Y -30.111,Z -92.298,A -90.000,B 90.000,C 0.000} C_DIS
LIN {X -55.289,Y -30.118,Z -92.118,A -90.000,B 90.000,C 0.000} C_DIS
LIN {X -55.410,Y -30.127,Z -91.903,A -90.000,B 90.000,C 0.000} C_DIS
LIN {X -56.358,Y -30.212,Z -90.190,A -90.000,B 90.000,C 0.000} C_DIS
LIN {X -56.905,Y -30.262,Z -89.198,A -90.000,B 90.000,C 0.000} C_DIS
LIN {X -57.297,Y -30.310,Z -88.499,A -90.000,B 90.000,C 0.000} C_DIS
LIN {X -57.335,Y -30.313,Z -88.433,A -90.000,B 90.000,C 0.000} C_DIS
LIN {X -58.046,Y -30.354,Z -87.179,A -90.000,B 90.000,C 0.000} C_DIS
LIN {X -58.118,Y -30.353,Z -87.047,A -90.000,B 90.000,C 0.000} C_DIS
LIN {X -58.193,Y -30.357,Z -86.895,A -90.000,B 90.000,C 0.000} C_DIS
LIN {X -58.512,Y -30.388,Z -86.190,A -90.000,B 90.000,C 0.000} C_DIS
LIN {X -58.686,Y -30.413,Z -85.815,A -90.000,B 90.000,C 0.000} C_DIS
LIN {X -58.896,Y -30.449,Z -85.339,A -90.000,B 90.000,C 0.000} C_DIS
LIN {X -58.923,Y -30.454,Z -85.279,A -90.000,B 90.000,C 0.000} C_DIS
LIN {X -58.989,Y -30.460,Z -85.147,A -90.000,B 90.000,C 0.000} C_DIS
LIN {X -59.483,Y -30.523,Z -84.173,A -90.000,B 90.000,C 0.000} C_DIS
LIN {X -59.882,Y -30.564,Z -83.400,A -90.000,B 90.000,C 0.000} C_DIS
LIN {X -59.922,Y -30.571,Z -83.325,A -90.000,B 90.000,C 0.000} C_DIS
LIN {X -59.993,Y -30.575,Z -83.185,A -90.000,B 90.000,C 0.000} C_DIS
LIN {X -60.040,Y -30.579,Z -83.086,A -90.000,B 90.000,C 0.000} C_DIS
LIN {X -60.086,Y -30.586,Z -82.974,A -90.000,B 90.000,C 0.000} C_DIS
LIN {X -60.253,Y -30.617,Z -82.547,A -90.000,B 90.000,C 0.000} C_DIS
LIN {X -60.337,Y -30.632,Z -82.319,A -90.000,B 90.000,C 0.000} C_DIS
LIN {X -60.429,Y -30.646,Z -82.068,A -90.000,B 90.000,C 0.000} C_DIS
LIN {X -60.626,Y -30.663,Z -81.610,A -90.000,B 90.000,C 0.000} C_DIS
LIN {X -60.836,Y -30.687,Z -81.131,A -90.000,B 90.000,C 0.000} C_DIS
LIN {X -61.182,Y -30.724,Z -80.363,A -90.000,B 90.000,C 0.000} C_DIS
LIN {X -61.228,Y -30.731,Z -80.261,A -90.000,B 90.000,C 0.000} C_DIS
LIN {X -61.317,Y -30.739,Z -80.044,A -90.000,B 90.000,C 0.000} C_DIS
LIN {X -61.401,Y -30.743,Z -79.832,A -90.000,B 90.000,C 0.000} C_DIS
LIN {X -61.640,Y -30.759,Z -79.194,A -90.000,B 90.000,C 0.000} C_DIS
LIN {X -61.789,Y -30.762,Z -78.841,A -90.000,B 90.000,C 0.000} C_DIS
LIN {X -61.935,Y -30.769,Z -78.509,A -90.000,B 90.000,C 0.000} C_DIS
LIN {X -61.983,Y -30.773,Z -78.392,A -90.000,B 90.000,C 0.000} C_DIS
LIN {X -62.268,Y -30.802,Z -77.625,A -90.000,B 90.000,C 0.000} C_DIS
LIN {X -62.382,Y -30.808,Z -77.307,A -90.000,B 90.000,C 0.000} C_DIS
LIN {X -62.638,Y -30.823,Z -76.565,A -90.000,B 90.000,C 0.000} C_DIS
LIN {X -62.769,Y -30.842,Z -76.145,A -90.000,B 90.000,C 0.000} C_DIS
LIN {X -62.938,Y -30.854,Z -75.528,A -90.000,B 90.000,C 0.000} C_DIS
LIN {X -63.062,Y -30.869,Z -75.075,A -90.000,B 90.000,C 0.000} C_DIS
LIN {X -63.125,Y -30.874,Z -74.859,A -90.000,B 90.000,C 0.000} C_DIS
LIN {X -63.313,Y -30.878,Z -74.220,A -90.000,B 90.000,C 0.000} C_DIS
LIN {X -63.522,Y -30.880,Z -73.588,A -90.000,B 90.000,C 0.000} C_DIS
LIN {X -63.563,Y -30.880,Z -73.463,A -90.000,B 90.000,C 0.000} C_DIS
LIN {X -63.740,Y -30.876,Z -73.031,A -90.000,B 90.000,C 0.000} C_DIS
LIN {X -63.902,Y -30.877,Z -72.575,A -90.000,B 90.000,C 0.000} C_DIS
LIN {X -64.215,Y -30.871,Z -71.916,A -90.000,B 90.000,C 0.000} C_DIS
LIN {X -64.250,Y -30.870,Z -71.839,A -90.000,B 90.000,C 0.000} C_DIS
LIN {X -64.321,Y -30.877,Z -71.656,A -90.000,B 90.000,C 0.000} C_DIS
LIN {X -64.455,Y -30.879,Z -71.404,A -90.000,B 90.000,C 0.000} C_DIS
LIN {X -64.665,Y -30.876,Z -71.007,A -90.000,B 90.000,C 0.000} C_DIS
LIN {X -64.801,Y -30.877,Z -70.781,A -90.000,B 90.000,C 0.000} C_DIS
LIN {X -65.114,Y -30.884,Z -70.234,A -90.000,B 90.000,C 0.000} C_DIS
LIN {X -65.203,Y -30.880,Z -70.118,A -90.000,B 90.000,C 0.000} C_DIS
LIN {X -65.758,Y -30.874,Z -69.391,A -90.000,B 90.000,C 0.000} C_DIS
LIN {X -65.889,Y -30.878,Z -69.218,A -90.000,B 90.000,C 0.000} C_DIS
LIN {X -66.316,Y -30.890,Z -68.580,A -90.000,B 90.000,C 0.000} C_DIS
LIN {X -66.415,Y -30.897,Z -68.434,A -90.000,B 90.000,C 0.000} C_DIS
LIN {X -67.132,Y -30.940,Z -67.431,A -90.000,B 90.000,C 0.000} C_DIS
LIN {X -67.207,Y -30.942,Z -67.325,A -90.000,B 90.000,C 0.000} C_DIS
LIN {X -67.305,Y -30.947,Z -67.174,A -90.000,B 90.000,C 0.000} C_DIS
LIN {X -67.361,Y -30.952,Z -67.071,A -90.000,B 90.000,C 0.000} C_DIS
LIN {X -67.413,Y -30.958,Z -66.960,A -90.000,B 90.000,C 0.000} C_DIS
LIN {X -67.564,Y -30.982,Z -66.590,A -90.000,B 90.000,C 0.000} C_DIS
LIN {X -67.670,Y -31.003,Z -66.302,A -90.000,B 90.000,C 0.000} C_DIS
LIN {X -67.729,Y -31.023,Z -66.083,A -90.000,B 90.000,C 0.000} C_DIS
LIN {X -67.754,Y -31.034,Z -65.970,A -90.000,B 90.000,C 0.000} C_DIS
LIN {X -67.812,Y -31.050,Z -65.698,A -90.000,B 90.000,C 0.000} C_DIS
LIN {X -67.849,Y -31.055,Z -65.520,A -90.000,B 90.000,C 0.000} C_DIS
LIN {X -67.886,Y -31.064,Z -65.241,A -90.000,B 90.000,C 0.000} C_DIS
LIN {X -67.901,Y -31.075,Z -65.013,A -90.000,B 90.000,C 0.000} C_DIS
LIN {X -67.900,Y -31.081,Z -64.852,A -90.000,B 90.000,C 0.000} C_DIS
LIN {X -67.895,Y -31.082,Z -64.774,A -90.000,B 90.000,C 0.000} C_DIS
LIN {X -67.885,Y -31.084,Z -64.676,A -90.000,B 90.000,C 0.000} C_DIS
LIN {X -67.853,Y -31.084,Z -64.500,A -90.000,B 90.000,C 0.000} C_DIS
LIN {X -67.816,Y -31.081,Z -64.338,A -90.000,B 90.000,C 0.000} C_DIS
LIN {X -67.778,Y -31.077,Z -64.194,A -90.000,B 90.000,C 0.000} C_DIS
LIN {X -67.757,Y -31.076,Z -64.128,A -90.000,B 90.000,C 0.000} C_DIS
LIN {X -67.625,Y -31.071,Z -63.828,A -90.000,B 90.000,C 0.000} C_DIS
LIN {X -67.471,Y -31.070,Z -63.543,A -90.000,B 90.000,C 0.000} C_DIS
LIN {X -67.398,Y -31.064,Z -63.409,A -90.000,B 90.000,C 0.000} C_DIS
LIN {X -67.341,Y -31.054,Z -63.309,A -90.000,B 90.000,C 0.000} C_DIS
LIN {X -67.303,Y -31.047,Z -63.248,A -90.000,B 90.000,C 0.000} C_DIS
LIN {X -67.225,Y -31.035,Z -63.138,A -90.000,B 90.000,C 0.000} C_DIS
LIN {X -67.116,Y -31.022,Z -63.006,A -90.000,B 90.000,C 0.000} C_DIS
LIN {X -66.847,Y -30.984,Z -62.693,A -90.000,B 90.000,C 0.000} C_DIS
LIN {X -66.705,Y -30.964,Z -62.530,A -90.000,B 90.000,C 0.000} C_DIS
LIN {X -66.578,Y -30.948,Z -62.396,A -90.000,B 90.000,C 0.000} C_DIS
LIN {X -66.434,Y -30.933,Z -62.254,A -90.000,B 90.000,C 0.000} C_DIS
LIN {X -66.360,Y -30.926,Z -62.188,A -90.000,B 90.000,C 0.000} C_DIS
LIN {X -66.211,Y -30.915,Z -62.073,A -90.000,B 90.000,C 0.000} C_DIS
LIN {X -66.065,Y -30.899,Z -61.982,A -90.000,B 90.000,C 0.000} C_DIS
LIN {X -65.880,Y -30.883,Z -61.881,A -90.000,B 90.000,C 0.000} C_DIS
LIN {X -65.800,Y -30.876,Z -61.839,A -90.000,B 90.000,C 0.000} C_DIS
LIN {X -65.413,Y -30.848,Z -61.649,A -90.000,B 90.000,C 0.000} C_DIS
LIN {X -65.175,Y -30.833,Z -61.538,A -90.000,B 90.000,C 0.000} C_DIS
LIN {X -64.980,Y -30.821,Z -61.451,A -90.000,B 90.000,C 0.000} C_DIS
LIN {X -64.789,Y -30.813,Z -61.377,A -90.000,B 90.000,C 0.000} C_DIS
LIN {X -64.091,Y -30.793,Z -61.146,A -90.000,B 90.000,C 0.000} C_DIS
LIN {X -63.211,Y -30.760,Z -60.849,A -90.000,B 90.000,C 0.000} C_DIS
LIN {X -62.614,Y -30.729,Z -60.650,A -90.000,B 90.000,C 0.000} C_DIS
LIN {X -62.408,Y -30.722,Z -60.593,A -90.000,B 90.000,C 0.000} C_DIS
LIN {X -61.620,Y -30.709,Z -60.418,A -90.000,B 90.000,C 0.000} C_DIS
LIN {X -61.223,Y -30.706,Z -60.339,A -90.000,B 90.000,C 0.000} C_DIS
LIN {X -60.703,Y -30.696,Z -60.238,A -90.000,B 90.000,C 0.000} C_DIS
LIN {X -58.626,Y -30.672,Z -59.874,A -90.000,B 90.000,C 0.000} C_DIS
LIN {X -57.997,Y -30.667,Z -59.771,A -90.000,B 90.000,C 0.000} C_DIS
LIN {X -56.556,Y -30.647,Z -59.537,A -90.000,B 90.000,C 0.000} C_DIS
LIN {X -56.338,Y -30.646,Z -59.508,A -90.000,B 90.000,C 0.000} C_DIS
LIN {X -55.925,Y -30.649,Z -59.451,A -90.000,B 90.000,C 0.000} C_DIS
LIN {X -54.871,Y -30.648,Z -59.306,A -90.000,B 90.000,C 0.000} C_DIS
LIN {X -54.011,Y -30.653,Z -59.185,A -90.000,B 90.000,C 0.000} C_DIS
LIN {X -53.486,Y -30.654,Z -59.112,A -90.000,B 90.000,C 0.000} C_DIS
LIN {X -53.013,Y -30.651,Z -59.045,A -90.000,B 90.000,C 0.000} C_DIS
LIN {X -52.548,Y -30.654,Z -58.976,A -90.000,B 90.000,C 0.000} C_DIS
LIN {X -52.109,Y -30.651,Z -58.909,A -90.000,B 90.000,C 0.000} C_DIS
LIN {X -51.272,Y -30.661,Z -58.782,A -90.000,B 90.000,C 0.000} C_DIS
LIN {X -50.202,Y -30.655,Z -58.628,A -90.000,B 90.000,C 0.000} C_DIS
LIN {X -50.014,Y -30.658,Z -58.600,A -90.000,B 90.000,C 0.000} C_DIS
LIN {X -49.902,Y -30.657,Z -58.584,A -90.000,B 90.000,C 0.000} C_DIS
LIN {X -49.527,Y -30.664,Z -58.527,A -90.000,B 90.000,C 0.000} C_DIS
LIN {X -48.433,Y -30.682,Z -58.342,A -90.000,B 90.000,C 0.000} C_DIS
LIN {X -48.235,Y -30.682,Z -58.310,A -90.000,B 90.000,C 0.000} C_DIS
LIN {X -47.652,Y -30.676,Z -58.202,A -90.000,B 90.000,C 0.000} C_DIS
LIN {X -47.151,Y -30.676,Z -58.108,A -90.000,B 90.000,C 0.000} C_DIS
LIN {X -46.973,Y -30.675,Z -58.076,A -90.000,B 90.000,C 0.000} C_DIS
LIN {X -46.691,Y -30.673,Z -58.033,A -90.000,B 90.000,C 0.000} C_DIS
LIN {X -46.573,Y -30.672,Z -58.015,A -90.000,B 90.000,C 0.000} C_DIS
LIN {X -46.118,Y -30.649,Z -57.954,A -90.000,B 90.000,C 0.000} C_DIS
LIN {X -45.423,Y -30.628,Z -57.855,A -90.000,B 90.000,C 0.000} C_DIS
LIN {X -44.913,Y -30.597,Z -57.788,A -90.000,B 90.000,C 0.000} C_DIS
LIN {X -44.678,Y -30.586,Z -57.764,A -90.000,B 90.000,C 0.000} C_DIS
LIN {X -44.447,Y -30.568,Z -57.745,A -90.000,B 90.000,C 0.000} C_DIS
LIN {X -44.060,Y -30.535,Z -57.730,A -90.000,B 90.000,C 0.000} C_DIS
LIN {X -42.918,Y -30.445,Z -57.675,A -90.000,B 90.000,C 0.000} C_DIS
LIN {X -42.752,Y -30.432,Z -57.668,A -90.000,B 90.000,C 0.000} C_DIS
LIN {X -42.288,Y -30.407,Z -57.665,A -90.000,B 90.000,C 0.000} C_DIS
LIN {X -42.145,Y -30.389,Z -57.665,A -90.000,B 90.000,C 0.000} C_DIS
LIN {X -42.011,Y -30.373,Z -57.666,A -90.000,B 90.000,C 0.000} C_DIS
LIN {X -41.953,Y -30.367,Z -57.668,A -90.000,B 90.000,C 0.000} C_DIS
LIN {X -41.828,Y -30.357,Z -57.677,A -90.000,B 90.000,C 0.000} C_DIS
LIN {X -41.167,Y -30.318,Z -57.743,A -90.000,B 90.000,C 0.000} C_DIS
LIN {X -40.175,Y -30.248,Z -57.851,A -90.000,B 90.000,C 0.000} C_DIS
LIN {X -39.821,Y -30.219,Z -57.884,A -90.000,B 90.000,C 0.000} C_DIS
LIN {X -39.183,Y -30.173,Z -57.956,A -90.000,B 90.000,C 0.000} C_DIS
LIN {X -38.826,Y -30.142,Z -58.003,A -90.000,B 90.000,C 0.000} C_DIS
LIN {X -38.629,Y -30.126,Z -58.030,A -90.000,B 90.000,C 0.000} C_DIS
LIN {X -38.504,Y -30.119,Z -58.051,A -90.000,B 90.000,C 0.000} C_DIS
LIN {X -37.559,Y -30.088,Z -58.238,A -90.000,B 90.000,C 0.000} C_DIS
LIN {X -37.165,Y -30.077,Z -58.321,A -90.000,B 90.000,C 0.000} C_DIS
LIN {X -35.855,Y -30.052,Z -58.607,A -90.000,B 90.000,C 0.000} C_DIS
LIN {X -34.314,Y -30.011,Z -58.930,A -90.000,B 90.000,C 0.000} C_DIS
LIN {X -32.241,Y -29.994,Z -59.411,A -90.000,B 90.000,C 0.000} C_DIS
LIN {X -31.987,Y -29.993,Z -59.471,A -90.000,B 90.000,C 0.000} C_DIS
LIN {X -30.666,Y -30.003,Z -59.770,A -90.000,B 90.000,C 0.000} C_DIS
LIN {X -30.392,Y -30.006,Z -59.831,A -90.000,B 90.000,C 0.000} C_DIS
LIN {X -29.485,Y -30.034,Z -60.018,A -90.000,B 90.000,C 0.000} C_DIS
LIN {X -27.890,Y -30.105,Z -60.354,A -90.000,B 90.000,C 0.000} C_DIS
LIN {X -27.512,Y -30.124,Z -60.433,A -90.000,B 90.000,C 0.000} C_DIS
LIN {X -27.255,Y -30.136,Z -60.483,A -90.000,B 90.000,C 0.000} C_DIS
LIN {X -26.951,Y -30.156,Z -60.539,A -90.000,B 90.000,C 0.000} C_DIS
LIN {X -26.384,Y -30.196,Z -60.654,A -90.000,B 90.000,C 0.000} C_DIS
LIN {X -25.365,Y -30.255,Z -60.832,A -90.000,B 90.000,C 0.000} C_DIS
LIN {X -25.043,Y -30.287,Z -60.881,A -90.000,B 90.000,C 0.000} C_DIS
LIN {X -24.159,Y -30.350,Z -60.961,A -90.000,B 90.000,C 0.000} C_DIS
LIN {X -24.009,Y -30.280,Z -60.812,A -90.000,B 90.000,C 0.000} C_DIS
LIN {X -23.881,Y -30.233,Z -60.691,A -90.000,B 90.000,C 0.000} C_DIS
LIN {X -23.783,Y -30.201,Z -60.606,A -90.000,B 90.000,C 0.000} C_DIS
LIN {X -23.448,Y -30.096,Z -60.333,A -90.000,B 90.000,C 0.000} C_DIS
LIN {X -23.204,Y -30.019,Z -60.142,A -90.000,B 90.000,C 0.000} C_DIS
LIN {X -23.189,Y -30.015,Z -60.131,A -90.000,B 90.000,C 0.000} C_DIS
LIN {X -23.128,Y -30.001,Z -60.079,A -90.000,B 90.000,C 0.000} C_DIS
LIN {X -22.899,Y -29.945,Z -59.896,A -90.000,B 90.000,C 0.000} C_DIS
LIN {X -22.853,Y -29.934,Z -59.861,A -90.000,B 90.000,C 0.000} C_DIS
LIN {X -22.717,Y -29.908,Z -59.767,A -90.000,B 90.000,C 0.000} C_DIS
LIN {X -22.529,Y -29.877,Z -59.643,A -90.000,B 90.000,C 0.000} C_DIS
LIN {X -22.350,Y -29.861,Z -59.510,A -90.000,B 90.000,C 0.000} C_DIS
LIN {X -22.163,Y -29.848,Z -59.381,A -90.000,B 90.000,C 0.000} C_DIS
LIN {X -21.988,Y -29.836,Z -59.265,A -90.000,B 90.000,C 0.000} C_DIS
LIN {X -21.937,Y -29.832,Z -59.233,A -90.000,B 90.000,C 0.000} C_DIS
LIN {X -21.317,Y -29.810,Z -58.809,A -90.000,B 90.000,C 0.000} C_DIS
LIN {X -20.967,Y -29.797,Z -58.584,A -90.000,B 90.000,C 0.000} C_DIS
LIN {X -20.849,Y -29.797,Z -58.513,A -90.000,B 90.000,C 0.000} C_DIS
LIN {X -20.629,Y -29.803,Z -58.387,A -90.000,B 90.000,C 0.000} C_DIS
LIN {X -19.931,Y -29.813,Z -58.017,A -90.000,B 90.000,C 0.000} C_DIS
LIN {X -19.609,Y -29.828,Z -57.857,A -90.000,B 90.000,C 0.000} C_DIS
LIN {X -19.377,Y -29.837,Z -57.746,A -90.000,B 90.000,C 0.000} C_DIS
LIN {X -19.076,Y -29.853,Z -57.608,A -90.000,B 90.000,C 0.000} C_DIS
LIN {X -18.450,Y -29.898,Z -57.332,A -90.000,B 90.000,C 0.000} C_DIS
LIN {X -17.265,Y -29.928,Z -56.873,A -90.000,B 90.000,C 0.000} C_DIS
LIN {X -16.667,Y -29.945,Z -56.644,A -90.000,B 90.000,C 0.000} C_DIS
LIN {X -16.578,Y -29.948,Z -56.611,A -90.000,B 90.000,C 0.000} C_DIS
LIN {X -16.439,Y -29.957,Z -56.565,A -90.000,B 90.000,C 0.000} C_DIS
LIN {X -15.849,Y -29.995,Z -56.392,A -90.000,B 90.000,C 0.000} C_DIS
LIN {X -15.518,Y -29.999,Z -56.312,A -90.000,B 90.000,C 0.000} C_DIS
LIN {X -15.184,Y -30.004,Z -56.237,A -90.000,B 90.000,C 0.000} C_DIS
LIN {X -15.049,Y -30.009,Z -56.211,A -90.000,B 90.000,C 0.000} C_DIS
LIN {X -14.977,Y -30.013,Z -56.198,A -90.000,B 90.000,C 0.000} C_DIS
LIN {X -14.296,Y -30.028,Z -56.098,A -90.000,B 90.000,C 0.000} C_DIS
LIN {X -13.962,Y -30.042,Z -56.058,A -90.000,B 90.000,C 0.000} C_DIS
LIN {X -13.605,Y -30.059,Z -56.021,A -90.000,B 90.000,C 0.000} C_DIS
LIN {X -13.159,Y -30.082,Z -55.978,A -90.000,B 90.000,C 0.000} C_DIS
LIN {X -12.736,Y -30.109,Z -55.934,A -90.000,B 90.000,C 0.000} C_DIS
LIN {X -12.430,Y -30.120,Z -55.910,A -90.000,B 90.000,C 0.000} C_DIS
LIN {X -12.105,Y -30.137,Z -55.892,A -90.000,B 90.000,C 0.000} C_DIS
LIN {X -11.889,Y -30.144,Z -55.883,A -90.000,B 90.000,C 0.000} C_DIS
LIN {X -11.819,Y -30.143,Z -55.883,A -90.000,B 90.000,C 0.000} C_DIS
LIN {X -11.530,Y -30.148,Z -55.890,A -90.000,B 90.000,C 0.000} C_DIS
LIN {X -11.076,Y -30.146,Z -55.913,A -90.000,B 90.000,C 0.000} C_DIS
LIN {X -10.628,Y -30.144,Z -55.949,A -90.000,B 90.000,C 0.000} C_DIS
LIN {X -9.395,Y -30.181,Z -56.074,A -90.000,B 90.000,C 0.000} C_DIS
LIN {X -9.296,Y -30.186,Z -56.087,A -90.000,B 90.000,C 0.000} C_DIS
LIN {X -8.950,Y -30.208,Z -56.136,A -90.000,B 90.000,C 0.000} C_DIS
LIN {X -8.311,Y -30.213,Z -56.249,A -90.000,B 90.000,C 0.000} C_DIS
LIN {X -7.747,Y -30.212,Z -56.355,A -90.000,B 90.000,C 0.000} C_DIS
LIN {X -7.004,Y -30.202,Z -56.509,A -90.000,B 90.000,C 0.000} C_DIS
LIN {X -6.621,Y -30.202,Z -56.595,A -90.000,B 90.000,C 0.000} C_DIS
LIN {X -5.558,Y -30.213,Z -56.857,A -90.000,B 90.000,C 0.000} C_DIS
LIN {X -5.370,Y -30.212,Z -56.905,A -90.000,B 90.000,C 0.000} C_DIS
LIN {X -4.667,Y -30.200,Z -57.091,A -90.000,B 90.000,C 0.000} C_DIS
LIN {X -3.652,Y -30.168,Z -57.337,A -90.000,B 90.000,C 0.000} C_DIS
LIN {X -3.219,Y -30.163,Z -57.457,A -90.000,B 90.000,C 0.000} C_DIS
LIN {X -2.868,Y -30.164,Z -57.550,A -90.000,B 90.000,C 0.000} C_DIS
LIN {X -1.858,Y -30.149,Z -57.832,A -90.000,B 90.000,C 0.000} C_DIS
LIN {X -1.144,Y -30.117,Z -57.999,A -90.000,B 90.000,C 0.000} C_DIS
LIN {X -0.670,Y -30.105,Z -58.124,A -90.000,B 90.000,C 0.000} C_DIS
LIN {X -0.491,Y -30.106,Z -58.168,A -90.000,B 90.000,C 0.000} C_DIS
LIN {X 0.889,Y -30.092,Z -58.521,A -90.000,B 90.000,C 0.000} C_DIS
LIN {X 0.969,Y -30.091,Z -58.541,A -90.000,B 90.000,C 0.000} C_DIS
LIN {X 2.054,Y -30.053,Z -58.772,A -90.000,B 90.000,C 0.000} C_DIS
LIN {X 2.890,Y -30.051,Z -58.929,A -90.000,B 90.000,C 0.000} C_DIS
LIN {X 3.315,Y -30.045,Z -59.001,A -90.000,B 90.000,C 0.000} C_DIS
LIN {X 3.577,Y -30.039,Z -59.043,A -90.000,B 90.000,C 0.000} C_DIS
LIN {X 4.235,Y -30.031,Z -59.140,A -90.000,B 90.000,C 0.000} C_DIS
LIN {X 5.425,Y -30.037,Z -59.290,A -90.000,B 90.000,C 0.000} C_DIS
LIN {X 5.662,Y -30.037,Z -59.311,A -90.000,B 90.000,C 0.000} C_DIS
LIN {X 6.379,Y -30.034,Z -59.368,A -90.000,B 90.000,C 0.000} C_DIS
LIN {X 6.726,Y -30.039,Z -59.390,A -90.000,B 90.000,C 0.000} C_DIS
LIN {X 7.423,Y -30.058,Z -59.426,A -90.000,B 90.000,C 0.000} C_DIS
LIN {X 7.992,Y -30.057,Z -59.432,A -90.000,B 90.000,C 0.000} C_DIS
LIN {X 8.336,Y -30.064,Z -59.430,A -90.000,B 90.000,C 0.000} C_DIS
LIN {X 8.757,Y -30.076,Z -59.426,A -90.000,B 90.000,C 0.000} C_DIS
LIN {X 9.453,Y -30.066,Z -59.377,A -90.000,B 90.000,C 0.000} C_DIS
LIN {X 9.780,Y -30.069,Z -59.349,A -90.000,B 90.000,C 0.000} C_DIS
LIN {X 9.826,Y -30.070,Z -59.345,A -90.000,B 90.000,C 0.000} C_DIS
LIN {X 10.596,Y -30.045,Z -59.228,A -90.000,B 90.000,C 0.000} C_DIS
LIN {X 10.890,Y -30.020,Z -59.167,A -90.000,B 90.000,C 0.000} C_DIS
LIN {X 11.194,Y -30.003,Z -59.097,A -90.000,B 90.000,C 0.000} C_DIS
LIN {X 11.472,Y -29.976,Z -59.019,A -90.000,B 90.000,C 0.000} C_DIS
LIN {X 11.955,Y -29.915,Z -58.866,A -90.000,B 90.000,C 0.000} C_DIS
LIN {X 12.125,Y -29.889,Z -58.816,A -90.000,B 90.000,C 0.000} C_DIS
LIN {X 12.788,Y -29.823,Z -58.603,A -90.000,B 90.000,C 0.000} C_DIS
LIN {X 12.828,Y -29.818,Z -58.591,A -90.000,B 90.000,C 0.000} C_DIS
LIN {X 13.166,Y -29.797,Z -58.481,A -90.000,B 90.000,C 0.000} C_DIS
LIN {X 13.289,Y -29.793,Z -58.438,A -90.000,B 90.000,C 0.000} C_DIS
LIN {X 13.604,Y -29.785,Z -58.339,A -90.000,B 90.000,C 0.000} C_DIS
LIN {X 13.833,Y -29.783,Z -58.273,A -90.000,B 90.000,C 0.000} C_DIS
LIN {X 14.155,Y -29.780,Z -58.185,A -90.000,B 90.000,C 0.000} C_DIS
LIN {X 14.245,Y -29.775,Z -58.166,A -90.000,B 90.000,C 0.000} C_DIS
LIN {X 14.560,Y -29.775,Z -58.084,A -90.000,B 90.000,C 0.000} C_DIS
LIN {X 14.850,Y -29.790,Z -58.021,A -90.000,B 90.000,C 0.000} C_DIS
LIN {X 14.881,Y -29.792,Z -58.015,A -90.000,B 90.000,C 0.000} C_DIS
LIN {X 15.075,Y -29.792,Z -57.987,A -90.000,B 90.000,C 0.000} C_DIS
LIN {X 15.273,Y -29.796,Z -57.963,A -90.000,B 90.000,C 0.000} C_DIS
LIN {X 15.371,Y -29.794,Z -57.953,A -90.000,B 90.000,C 0.000} C_DIS
LIN {X 15.605,Y -29.797,Z -57.919,A -90.000,B 90.000,C 0.000} C_DIS
LIN {X 15.811,Y -29.800,Z -57.892,A -90.000,B 90.000,C 0.000} C_DIS
LIN {X 15.956,Y -29.809,Z -57.878,A -90.000,B 90.000,C 0.000} C_DIS
LIN {X 16.284,Y -29.809,Z -57.870,A -90.000,B 90.000,C 0.000} C_DIS
LIN {X 16.379,Y -29.810,Z -57.870,A -90.000,B 90.000,C 0.000} C_DIS
LIN {X 16.622,Y -29.811,Z -57.891,A -90.000,B 90.000,C 0.000} C_DIS
LIN {X 16.873,Y -29.825,Z -57.899,A -90.000,B 90.000,C 0.000} C_DIS
LIN {X 16.989,Y -29.834,Z -57.905,A -90.000,B 90.000,C 0.000} C_DIS
LIN {X 17.049,Y -29.837,Z -57.913,A -90.000,B 90.000,C 0.000} C_DIS
LIN {X 17.409,Y -29.837,Z -57.948,A -90.000,B 90.000,C 0.000} C_DIS
LIN {X 17.581,Y -29.829,Z -57.977,A -90.000,B 90.000,C 0.000} C_DIS
LIN {X 17.828,Y -29.828,Z -58.030,A -90.000,B 90.000,C 0.000} C_DIS
LIN {X 17.948,Y -29.825,Z -58.060,A -90.000,B 90.000,C 0.000} C_DIS
LIN {X 18.229,Y -29.753,Z -58.057,A -90.000,B 90.000,C 0.000} C_DIS
LIN {X 18.427,Y -29.709,Z -58.059,A -90.000,B 90.000,C 0.000} C_DIS
LIN {X 18.498,Y -29.689,Z -58.056,A -90.000,B 90.000,C 0.000} C_DIS
LIN {X 18.715,Y -29.625,Z -58.069,A -90.000,B 90.000,C 0.000} C_DIS
LIN {X 18.889,Y -29.580,Z -58.084,A -90.000,B 90.000,C 0.000} C_DIS
LIN {X 19.039,Y -29.576,Z -58.038,A -90.000,B 90.000,C 0.000} C_DIS
LIN {X 19.304,Y -29.565,Z -57.963,A -90.000,B 90.000,C 0.000} C_DIS
LIN {X 19.329,Y -29.566,Z -57.956,A -90.000,B 90.000,C 0.000} C_DIS
LIN {X 19.398,Y -29.570,Z -57.928,A -90.000,B 90.000,C 0.000} C_DIS
LIN {X 19.700,Y -29.582,Z -57.824,A -90.000,B 90.000,C 0.000} C_DIS
LIN {X 19.957,Y -29.601,Z -57.742,A -90.000,B 90.000,C 0.000} C_DIS
LIN {X 20.240,Y -29.610,Z -57.678,A -90.000,B 90.000,C 0.000} C_DIS
LIN {X 20.395,Y -29.619,Z -57.646,A -90.000,B 90.000,C 0.000} C_DIS
LIN {X 20.745,Y -29.630,Z -57.603,A -90.000,B 90.000,C 0.000} C_DIS
LIN {X 20.870,Y -29.633,Z -57.590,A -90.000,B 90.000,C 0.000} C_DIS
LIN {X 21.039,Y -29.640,Z -57.581,A -90.000,B 90.000,C 0.000} C_DIS
LIN {X 21.306,Y -29.654,Z -57.571,A -90.000,B 90.000,C 0.000} C_DIS
LIN {X 21.510,Y -29.656,Z -57.581,A -90.000,B 90.000,C 0.000} C_DIS
LIN {X 21.602,Y -29.689,Z -57.547,A -90.000,B 90.000,C 0.000} C_DIS
LIN {X 21.763,Y -29.688,Z -57.439,A -90.000,B 90.000,C 0.000} C_DIS
LIN {X 22.383,Y -29.684,Z -57.069,A -90.000,B 90.000,C 0.000} C_DIS
LIN {X 22.841,Y -29.690,Z -56.807,A -90.000,B 90.000,C 0.000} C_DIS
LIN {X 23.171,Y -29.687,Z -56.631,A -90.000,B 90.000,C 0.000} C_DIS
LIN {X 23.247,Y -29.739,Z -56.513,A -90.000,B 90.000,C 0.000} C_DIS
LIN {X 23.358,Y -29.814,Z -56.352,A -90.000,B 90.000,C 0.000} C_DIS
LIN {X 23.436,Y -29.868,Z -56.248,A -90.000,B 90.000,C 0.000} C_DIS
LIN {X 23.443,Y -29.865,Z -56.194,A -90.000,B 90.000,C 0.000} C_DIS
LIN {X 23.507,Y -29.850,Z -55.843,A -90.000,B 90.000,C 0.000} C_DIS
LIN {X 23.536,Y -29.842,Z -55.694,A -90.000,B 90.000,C 0.000} C_DIS
LIN {X 23.587,Y -29.830,Z -55.521,A -90.000,B 90.000,C 0.000} C_DIS
LIN {X 23.646,Y -29.821,Z -55.329,A -90.000,B 90.000,C 0.000} C_DIS
LIN {X 23.742,Y -29.795,Z -55.084,A -90.000,B 90.000,C 0.000} C_DIS
LIN {X 23.789,Y -29.788,Z -54.977,A -90.000,B 90.000,C 0.000} C_DIS
LIN {X 23.909,Y -29.770,Z -54.720,A -90.000,B 90.000,C 0.000} C_DIS
LIN {X 24.056,Y -29.737,Z -54.458,A -90.000,B 90.000,C 0.000} C_DIS
LIN {X 24.118,Y -29.727,Z -54.357,A -90.000,B 90.000,C 0.000} C_DIS
LIN {X 24.222,Y -29.712,Z -54.201,A -90.000,B 90.000,C 0.000} C_DIS
LIN {X 24.359,Y -29.687,Z -54.011,A -90.000,B 90.000,C 0.000} C_DIS
LIN {X 24.437,Y -29.676,Z -53.907,A -90.000,B 90.000,C 0.000} C_DIS
LIN {X 24.466,Y -29.673,Z -53.869,A -90.000,B 90.000,C 0.000} C_DIS
LIN {X 24.741,Y -29.627,Z -53.569,A -90.000,B 90.000,C 0.000} C_DIS
LIN {X 24.881,Y -29.609,Z -53.429,A -90.000,B 90.000,C 0.000} C_DIS
LIN {X 25.187,Y -29.570,Z -53.153,A -90.000,B 90.000,C 0.000} C_DIS
LIN {X 25.315,Y -29.559,Z -53.049,A -90.000,B 90.000,C 0.000} C_DIS
LIN {X 25.550,Y -29.533,Z -52.877,A -90.000,B 90.000,C 0.000} C_DIS
LIN {X 25.716,Y -29.520,Z -52.758,A -90.000,B 90.000,C 0.000} C_DIS
LIN {X 25.797,Y -29.575,Z -52.548,A -90.000,B 90.000,C 0.000} C_DIS
LIN {X 25.857,Y -29.612,Z -52.410,A -90.000,B 90.000,C 0.000} C_DIS
LIN {X 25.898,Y -29.638,Z -52.325,A -90.000,B 90.000,C 0.000} C_DIS
LIN {X 25.955,Y -29.675,Z -52.218,A -90.000,B 90.000,C 0.000} C_DIS
LIN {X 26.068,Y -29.749,Z -52.015,A -90.000,B 90.000,C 0.000} C_DIS
LIN {X 26.172,Y -29.808,Z -51.853,A -90.000,B 90.000,C 0.000} C_DIS
LIN {X 26.231,Y -29.843,Z -51.768,A -90.000,B 90.000,C 0.000} C_DIS
LIN {X 26.284,Y -29.874,Z -51.695,A -90.000,B 90.000,C 0.000} C_DIS
LIN {X 26.289,Y -29.873,Z -51.666,A -90.000,B 90.000,C 0.000} C_DIS
LIN {X 26.315,Y -29.868,Z -51.535,A -90.000,B 90.000,C 0.000} C_DIS
LIN {X 26.351,Y -29.862,Z -51.381,A -90.000,B 90.000,C 0.000} C_DIS
LIN {X 26.444,Y -29.852,Z -51.054,A -90.000,B 90.000,C 0.000} C_DIS
LIN {X 26.559,Y -29.833,Z -50.682,A -90.000,B 90.000,C 0.000} C_DIS
LIN {X 26.628,Y -29.817,Z -50.482,A -90.000,B 90.000,C 0.000} C_DIS
LIN {X 26.661,Y -29.810,Z -50.394,A -90.000,B 90.000,C 0.000} C_DIS
LIN {X 26.869,Y -29.791,Z -49.912,A -90.000,B 90.000,C 0.000} C_DIS
LIN {X 26.938,Y -29.787,Z -49.762,A -90.000,B 90.000,C 0.000} C_DIS
LIN {X 27.120,Y -29.771,Z -49.387,A -90.000,B 90.000,C 0.000} C_DIS
LIN {X 27.182,Y -29.763,Z -49.272,A -90.000,B 90.000,C 0.000} C_DIS
LIN {X 27.439,Y -29.747,Z -48.830,A -90.000,B 90.000,C 0.000} C_DIS
LIN {X 27.518,Y -29.741,Z -48.706,A -90.000,B 90.000,C 0.000} C_DIS
LIN {X 27.668,Y -29.738,Z -48.482,A -90.000,B 90.000,C 0.000} C_DIS
LIN {X 27.755,Y -29.735,Z -48.349,A -90.000,B 90.000,C 0.000} C_DIS
LIN {X 27.918,Y -29.716,Z -48.136,A -90.000,B 90.000,C 0.000} C_DIS
LIN {X 28.015,Y -29.707,Z -48.012,A -90.000,B 90.000,C 0.000} C_DIS
LIN {X 28.122,Y -29.694,Z -47.885,A -90.000,B 90.000,C 0.000} C_DIS
LIN {X 28.245,Y -29.683,Z -47.733,A -90.000,B 90.000,C 0.000} C_DIS
LIN {X 28.458,Y -29.681,Z -47.486,A -90.000,B 90.000,C 0.000} C_DIS
LIN {X 28.568,Y -29.672,Z -47.375,A -90.000,B 90.000,C 0.000} C_DIS
LIN {X 28.663,Y -29.669,Z -47.283,A -90.000,B 90.000,C 0.000} C_DIS
LIN {X 28.768,Y -29.668,Z -47.184,A -90.000,B 90.000,C 0.000} C_DIS
LIN {X 28.950,Y -29.658,Z -47.029,A -90.000,B 90.000,C 0.000} C_DIS
LIN {X 29.150,Y -29.641,Z -46.855,A -90.000,B 90.000,C 0.000} C_DIS
LIN {X 29.201,Y -29.638,Z -46.811,A -90.000,B 90.000,C 0.000} C_DIS
LIN {X 29.582,Y -29.599,Z -46.539,A -90.000,B 90.000,C 0.000} C_DIS
LIN {X 29.622,Y -29.596,Z -46.511,A -90.000,B 90.000,C 0.000} C_DIS
LIN {X 29.826,Y -29.594,Z -46.360,A -90.000,B 90.000,C 0.000} C_DIS
LIN {X 30.091,Y -29.583,Z -46.183,A -90.000,B 90.000,C 0.000} C_DIS
LIN {X 30.197,Y -29.581,Z -46.114,A -90.000,B 90.000,C 0.000} C_DIS
LIN {X 30.620,Y -29.563,Z -45.884,A -90.000,B 90.000,C 0.000} C_DIS
LIN {X 30.693,Y -29.562,Z -45.846,A -90.000,B 90.000,C 0.000} C_DIS
LIN {X 31.118,Y -29.543,Z -45.654,A -90.000,B 90.000,C 0.000} C_DIS
LIN {X 31.420,Y -29.517,Z -45.548,A -90.000,B 90.000,C 0.000} C_DIS
LIN {X 31.856,Y -29.488,Z -45.402,A -90.000,B 90.000,C 0.000} C_DIS
LIN {X 32.312,Y -29.476,Z -45.258,A -90.000,B 90.000,C 0.000} C_DIS
LIN {X 32.427,Y -29.474,Z -45.222,A -90.000,B 90.000,C 0.000} C_DIS
LIN {X 32.974,Y -29.464,Z -45.102,A -90.000,B 90.000,C 0.000} C_DIS
LIN {X 33.438,Y -29.457,Z -45.025,A -90.000,B 90.000,C 0.000} C_DIS
LIN {X 33.818,Y -29.447,Z -44.987,A -90.000,B 90.000,C 0.000} C_DIS
LIN {X 34.068,Y -29.436,Z -44.966,A -90.000,B 90.000,C 0.000} C_DIS
LIN {X 34.576,Y -29.411,Z -44.941,A -90.000,B 90.000,C 0.000} C_DIS
LIN {X 35.194,Y -29.403,Z -44.916,A -90.000,B 90.000,C 0.000} C_DIS
LIN {X 35.321,Y -29.402,Z -44.912,A -90.000,B 90.000,C 0.000} C_DIS
LIN {X 35.675,Y -29.392,Z -44.926,A -90.000,B 90.000,C 0.000} C_DIS
LIN {X 35.961,Y -29.390,Z -44.943,A -90.000,B 90.000,C 0.000} C_DIS
LIN {X 36.875,Y -29.382,Z -45.010,A -90.000,B 90.000,C 0.000} C_DIS
LIN {X 37.267,Y -29.383,Z -45.039,A -90.000,B 90.000,C 0.000} C_DIS
LIN {X 37.509,Y -29.385,Z -45.055,A -90.000,B 90.000,C 0.000} C_DIS
LIN {X 38.230,Y -29.403,Z -45.105,A -90.000,B 90.000,C 0.000} C_DIS
LIN {X 38.898,Y -29.439,Z -45.099,A -90.000,B 90.000,C 0.000} C_DIS
LIN {X 39.486,Y -29.507,Z -45.015,A -90.000,B 90.000,C 0.000} C_DIS
LIN {X 39.639,Y -29.526,Z -44.993,A -90.000,B 90.000,C 0.000} C_DIS
LIN {X 40.107,Y -29.606,Z -44.902,A -90.000,B 90.000,C 0.000} C_DIS
LIN {X 40.507,Y -29.665,Z -44.817,A -90.000,B 90.000,C 0.000} C_DIS
LIN {X 41.018,Y -29.695,Z -44.673,A -90.000,B 90.000,C 0.000} C_DIS
LIN {X 41.659,Y -29.706,Z -44.472,A -90.000,B 90.000,C 0.000} C_DIS
LIN {X 42.156,Y -29.709,Z -44.321,A -90.000,B 90.000,C 0.000} C_DIS
LIN {X 42.615,Y -29.710,Z -44.183,A -90.000,B 90.000,C 0.000} C_DIS
LIN {X 43.000,Y -29.715,Z -44.073,A -90.000,B 90.000,C 0.000} C_DIS
LIN {X 43.417,Y -29.700,Z -43.983,A -90.000,B 90.000,C 0.000} C_DIS
LIN {X 43.741,Y -29.680,Z -43.924,A -90.000,B 90.000,C 0.000} C_DIS
LIN {X 44.205,Y -29.661,Z -43.826,A -90.000,B 90.000,C 0.000} C_DIS
LIN {X 44.273,Y -29.658,Z -43.812,A -90.000,B 90.000,C 0.000} C_DIS
LIN {X 44.383,Y -29.655,Z -43.790,A -90.000,B 90.000,C 0.000} C_DIS
LIN {X 44.850,Y -29.654,Z -43.704,A -90.000,B 90.000,C 0.000} C_DIS
LIN {X 45.186,Y -29.659,Z -43.649,A -90.000,B 90.000,C 0.000} C_DIS
LIN {X 45.824,Y -29.660,Z -43.598,A -90.000,B 90.000,C 0.000} C_DIS
LIN {X 46.399,Y -29.646,Z -43.580,A -90.000,B 90.000,C 0.000} C_DIS
LIN {X 46.708,Y -29.638,Z -43.574,A -90.000,B 90.000,C 0.000} C_DIS
LIN {X 47.317,Y -29.595,Z -43.606,A -90.000,B 90.000,C 0.000} C_DIS
LIN {X 47.419,Y -29.590,Z -43.613,A -90.000,B 90.000,C 0.000} C_DIS
LIN {X 47.916,Y -29.580,Z -43.653,A -90.000,B 90.000,C 0.000} C_DIS
LIN {X 48.034,Y -29.580,Z -43.664,A -90.000,B 90.000,C 0.000} C_DIS
LIN {X 48.565,Y -29.568,Z -43.737,A -90.000,B 90.000,C 0.000} C_DIS
LIN {X 49.008,Y -29.558,Z -43.821,A -90.000,B 90.000,C 0.000} C_DIS
LIN {X 49.089,Y -29.555,Z -43.839,A -90.000,B 90.000,C 0.000} C_DIS
LIN {X 49.332,Y -29.547,Z -43.892,A -90.000,B 90.000,C 0.000} C_DIS
LIN {X 49.630,Y -29.540,Z -43.966,A -90.000,B 90.000,C 0.000} C_DIS
LIN {X 49.806,Y -29.535,Z -44.011,A -90.000,B 90.000,C 0.000} C_DIS
LIN {X 50.118,Y -29.532,Z -44.091,A -90.000,B 90.000,C 0.000} C_DIS
LIN {X 50.847,Y -29.506,Z -44.318,A -90.000,B 90.000,C 0.000} C_DIS
LIN {X 51.021,Y -29.500,Z -44.377,A -90.000,B 90.000,C 0.000} C_DIS
LIN {X 51.284,Y -29.497,Z -44.469,A -90.000,B 90.000,C 0.000} C_DIS
LIN {X 51.815,Y -29.487,Z -44.671,A -90.000,B 90.000,C 0.000} C_DIS
LIN {X 51.935,Y -29.486,Z -44.717,A -90.000,B 90.000,C 0.000} C_DIS
LIN {X 52.148,Y -29.488,Z -44.801,A -90.000,B 90.000,C 0.000} C_DIS
LIN {X 52.573,Y -29.480,Z -45.002,A -90.000,B 90.000,C 0.000} C_DIS
LIN {X 53.379,Y -29.464,Z -45.408,A -90.000,B 90.000,C 0.000} C_DIS
LIN {X 53.886,Y -29.454,Z -45.681,A -90.000,B 90.000,C 0.000} C_DIS
LIN {X 54.450,Y -29.448,Z -45.986,A -90.000,B 90.000,C 0.000} C_DIS
LIN {X 54.950,Y -29.447,Z -46.264,A -90.000,B 90.000,C 0.000} C_DIS
LIN {X 55.320,Y -29.454,Z -46.474,A -90.000,B 90.000,C 0.000} C_DIS
LIN {X 55.443,Y -29.456,Z -46.551,A -90.000,B 90.000,C 0.000} C_DIS
LIN {X 55.716,Y -29.463,Z -46.730,A -90.000,B 90.000,C 0.000} C_DIS
LIN {X 56.225,Y -29.460,Z -47.111,A -90.000,B 90.000,C 0.000} C_DIS
LIN {X 57.905,Y -29.433,Z -48.420,A -90.000,B 90.000,C 0.000} C_DIS
LIN {X 58.118,Y -29.432,Z -48.587,A -90.000,B 90.000,C 0.000} C_DIS
LIN {X 58.303,Y -29.431,Z -48.736,A -90.000,B 90.000,C 0.000} C_DIS
LIN {X 58.488,Y -29.435,Z -48.887,A -90.000,B 90.000,C 0.000} C_DIS
LIN {X 59.435,Y -29.427,Z -49.745,A -90.000,B 90.000,C 0.000} C_DIS
LIN {X 60.584,Y -29.418,Z -50.780,A -90.000,B 90.000,C 0.000} C_DIS
LIN {X 60.680,Y -29.419,Z -50.867,A -90.000,B 90.000,C 0.000} C_DIS
LIN {X 62.215,Y -29.416,Z -52.328,A -90.000,B 90.000,C 0.000} C_DIS
LIN {X 62.759,Y -29.414,Z -52.843,A -90.000,B 90.000,C 0.000} C_DIS
LIN {X 63.966,Y -29.420,Z -53.934,A -90.000,B 90.000,C 0.000} C_DIS
LIN {X 64.112,Y -29.420,Z -54.067,A -90.000,B 90.000,C 0.000} C_DIS
LIN {X 64.796,Y -29.423,Z -54.691,A -90.000,B 90.000,C 0.000} C_DIS
LIN {X 65.271,Y -29.431,Z -55.072,A -90.000,B 90.000,C 0.000} C_DIS
LIN {X 65.956,Y -29.441,Z -55.617,A -90.000,B 90.000,C 0.000} C_DIS
LIN {X 66.625,Y -29.451,Z -56.136,A -90.000,B 90.000,C 0.000} C_DIS
LIN {X 68.694,Y -29.497,Z -57.698,A -90.000,B 90.000,C 0.000} C_DIS
LIN {X 69.145,Y -29.504,Z -58.045,A -90.000,B 90.000,C 0.000} C_DIS
LIN {X 70.220,Y -29.534,Z -58.879,A -90.000,B 90.000,C 0.000} C_DIS
LIN {X 70.456,Y -29.543,Z -59.068,A -90.000,B 90.000,C 0.000} C_DIS
LIN {X 70.965,Y -29.561,Z -59.487,A -90.000,B 90.000,C 0.000} C_DIS
LIN {X 71.467,Y -29.566,Z -59.935,A -90.000,B 90.000,C 0.000} C_DIS
LIN {X 71.758,Y -29.575,Z -60.202,A -90.000,B 90.000,C 0.000} C_DIS
LIN {X 72.940,Y -29.627,Z -61.341,A -90.000,B 90.000,C 0.000} C_DIS
LIN {X 73.175,Y -29.622,Z -61.604,A -90.000,B 90.000,C 0.000} C_DIS
LIN {X 73.515,Y -29.619,Z -61.988,A -90.000,B 90.000,C 0.000} C_DIS
LIN {X 73.990,Y -29.634,Z -62.550,A -90.000,B 90.000,C 0.000} C_DIS
LIN {X 74.619,Y -29.647,Z -63.293,A -90.000,B 90.000,C 0.000} C_DIS
LIN {X 74.779,Y -29.641,Z -63.506,A -90.000,B 90.000,C 0.000} C_DIS
LIN {X 74.925,Y -29.640,Z -63.703,A -90.000,B 90.000,C 0.000} C_DIS
LIN {X 75.033,Y -29.641,Z -63.849,A -90.000,B 90.000,C 0.000} C_DIS
LIN {X 75.215,Y -29.641,Z -64.109,A -90.000,B 90.000,C 0.000} C_DIS
LIN {X 75.821,Y -29.652,Z -64.984,A -90.000,B 90.000,C 0.000} C_DIS
LIN {X 75.874,Y -29.653,Z -65.063,A -90.000,B 90.000,C 0.000} C_DIS
LIN {X 75.992,Y -29.648,Z -65.231,A -90.000,B 90.000,C 0.000} C_DIS
LIN {X 76.295,Y -29.631,Z -65.696,A -90.000,B 90.000,C 0.000} C_DIS
LIN {X 76.450,Y -29.631,Z -65.944,A -90.000,B 90.000,C 0.000} C_DIS
LIN {X 76.508,Y -29.633,Z -66.030,A -90.000,B 90.000,C 0.000} C_DIS
LIN {X 76.955,Y -29.621,Z -66.665,A -90.000,B 90.000,C 0.000} C_DIS
LIN {X 77.128,Y -29.609,Z -66.937,A -90.000,B 90.000,C 0.000} C_DIS
LIN {X 77.571,Y -29.607,Z -67.589,A -90.000,B 90.000,C 0.000} C_DIS
LIN {X 77.652,Y -29.605,Z -67.715,A -90.000,B 90.000,C 0.000} C_DIS
LIN {X 77.719,Y -29.598,Z -67.814,A -90.000,B 90.000,C 0.000} C_DIS
LIN {X 77.846,Y -29.591,Z -67.991,A -90.000,B 90.000,C 0.000} C_DIS
LIN {X 78.053,Y -29.583,Z -68.292,A -90.000,B 90.000,C 0.000} C_DIS
LIN {X 78.101,Y -29.582,Z -68.364,A -90.000,B 90.000,C 0.000} C_DIS
LIN {X 78.227,Y -29.573,Z -68.542,A -90.000,B 90.000,C 0.000} C_DIS
LIN {X 78.289,Y -29.527,Z -68.589,A -90.000,B 90.000,C 0.000} C_DIS
LIN {X 78.372,Y -29.479,Z -68.658,A -90.000,B 90.000,C 0.000} C_DIS
LIN {X 78.466,Y -29.432,Z -68.742,A -90.000,B 90.000,C 0.000} C_DIS
LIN {X 78.539,Y -29.401,Z -68.813,A -90.000,B 90.000,C 0.000} C_DIS
LIN {X 78.632,Y -29.367,Z -68.913,A -90.000,B 90.000,C 0.000} C_DIS
LIN {X 78.665,Y -29.357,Z -68.950,A -90.000,B 90.000,C 0.000} C_DIS
LIN {X 78.741,Y -29.337,Z -69.038,A -90.000,B 90.000,C 0.000} C_DIS
LIN {X 78.775,Y -29.330,Z -69.079,A -90.000,B 90.000,C 0.000} C_DIS
LIN {X 78.884,Y -29.313,Z -69.217,A -90.000,B 90.000,C 0.000} C_DIS
LIN {X 78.939,Y -29.309,Z -69.290,A -90.000,B 90.000,C 0.000} C_DIS
LIN {X 79.016,Y -29.315,Z -68.759,A -90.000,B 90.000,C 0.000} C_DIS
LIN {X 79.108,Y -29.327,Z -68.234,A -90.000,B 90.000,C 0.000} C_DIS
LIN {X 79.168,Y -29.338,Z -67.902,A -90.000,B 90.000,C 0.000} C_DIS
LIN {X 79.279,Y -29.361,Z -67.305,A -90.000,B 90.000,C 0.000} C_DIS
LIN {X 79.344,Y -29.379,Z -66.970,A -90.000,B 90.000,C 0.000} C_DIS
LIN {X 79.537,Y -29.408,Z -66.290,A -90.000,B 90.000,C 0.000} C_DIS
LIN {X 79.779,Y -29.445,Z -65.482,A -90.000,B 90.000,C 0.000} C_DIS
LIN {X 79.936,Y -29.474,Z -64.970,A -90.000,B 90.000,C 0.000} C_DIS
LIN {X 80.029,Y -29.496,Z -64.683,A -90.000,B 90.000,C 0.000} C_DIS
LIN {X 80.556,Y -29.556,Z -63.411,A -90.000,B 90.000,C 0.000} C_DIS
LIN {X 80.741,Y -29.585,Z -62.986,A -90.000,B 90.000,C 0.000} C_DIS
LIN {X 80.823,Y -29.598,Z -62.805,A -90.000,B 90.000,C 0.000} C_DIS
LIN {X 81.071,Y -29.639,Z -62.285,A -90.000,B 90.000,C 0.000} C_DIS
LIN {X 81.619,Y -29.716,Z -61.196,A -90.000,B 90.000,C 0.000} C_DIS
LIN {X 81.713,Y -29.729,Z -61.020,A -90.000,B 90.000,C 0.000} C_DIS
LIN {X 82.065,Y -29.791,Z -60.408,A -90.000,B 90.000,C 0.000} C_DIS
LIN {X 82.354,Y -29.854,Z -59.891,A -90.000,B 90.000,C 0.000} C_DIS
LIN {X 82.708,Y -29.926,Z -59.284,A -90.000,B 90.000,C 0.000} C_DIS
LIN {X 82.969,Y -29.980,Z -58.840,A -90.000,B 90.000,C 0.000} C_DIS
LIN {X 83.019,Y -29.988,Z -58.760,A -90.000,B 90.000,C 0.000} C_DIS
LIN {X 83.090,Y -30.001,Z -58.652,A -90.000,B 90.000,C 0.000} C_DIS
LIN {X 83.315,Y -30.045,Z -58.325,A -90.000,B 90.000,C 0.000} C_DIS
LIN {X 83.694,Y -30.128,Z -57.773,A -90.000,B 90.000,C 0.000} C_DIS
LIN {X 84.152,Y -30.231,Z -57.118,A -90.000,B 90.000,C 0.000} C_DIS
LIN {X 84.434,Y -30.287,Z -56.729,A -90.000,B 90.000,C 0.000} C_DIS
LIN {X 84.627,Y -30.328,Z -56.478,A -90.000,B 90.000,C 0.000} C_DIS
LIN {X 84.773,Y -30.363,Z -56.290,A -90.000,B 90.000,C 0.000} C_DIS
LIN {X 85.218,Y -30.475,Z -55.745,A -90.000,B 90.000,C 0.000} C_DIS
LIN {X 85.577,Y -30.568,Z -55.314,A -90.000,B 90.000,C 0.000} C_DIS
LIN {X 86.025,Y -30.683,Z -54.785,A -90.000,B 90.000,C 0.000} C_DIS
LIN {X 86.034,Y -30.680,Z -54.727,A -90.000,B 90.000,C 0.000} C_DIS
LIN {X 86.254,Y -30.598,Z -53.730,A -90.000,B 90.000,C 0.000} C_DIS
LIN {X 86.280,Y -30.569,Z -53.520,A -90.000,B 90.000,C 0.000} C_DIS
LIN {X 86.389,Y -30.438,Z -52.791,A -90.000,B 90.000,C 0.000} C_DIS
LIN {X 86.413,Y -30.410,Z -52.643,A -90.000,B 90.000,C 0.000} C_DIS
LIN {X 86.431,Y -30.389,Z -52.537,A -90.000,B 90.000,C 0.000} C_DIS
LIN {X 86.449,Y -30.371,Z -52.444,A -90.000,B 90.000,C 0.000} C_DIS
LIN {X 86.492,Y -30.347,Z -52.278,A -90.000,B 90.000,C 0.000} C_DIS
LIN {X 86.584,Y -30.309,Z -51.963,A -90.000,B 90.000,C 0.000} C_DIS
LIN {X 86.741,Y -30.257,Z -51.468,A -90.000,B 90.000,C 0.000} C_DIS
LIN {X 86.792,Y -30.234,Z -51.297,A -90.000,B 90.000,C 0.000} C_DIS
LIN {X 86.894,Y -30.197,Z -50.993,A -90.000,B 90.000,C 0.000} C_DIS
LIN {X 86.947,Y -30.183,Z -50.848,A -90.000,B 90.000,C 0.000} C_DIS
LIN {X 87.071,Y -30.161,Z -50.542,A -90.000,B 90.000,C 0.000} C_DIS
LIN {X 87.182,Y -30.140,Z -50.273,A -90.000,B 90.000,C 0.000} C_DIS
LIN {X 87.232,Y -30.127,Z -50.158,A -90.000,B 90.000,C 0.000} C_DIS
LIN {X 87.327,Y -30.101,Z -49.952,A -90.000,B 90.000,C 0.000} C_DIS
LIN {X 87.494,Y -30.063,Z -49.602,A -90.000,B 90.000,C 0.000} C_DIS
LIN {X 87.669,Y -30.037,Z -49.266,A -90.000,B 90.000,C 0.000} C_DIS
LIN {X 87.847,Y -30.002,Z -48.947,A -90.000,B 90.000,C 0.000} C_DIS
LIN {X 88.182,Y -29.944,Z -48.363,A -90.000,B 90.000,C 0.000} C_DIS
LIN {X 88.415,Y -29.911,Z -47.970,A -90.000,B 90.000,C 0.000} C_DIS
LIN {X 88.780,Y -29.831,Z -47.432,A -90.000,B 90.000,C 0.000} C_DIS
LIN {X 89.118,Y -29.779,Z -46.957,A -90.000,B 90.000,C 0.000} C_DIS
LIN {X 89.180,Y -29.770,Z -46.870,A -90.000,B 90.000,C 0.000} C_DIS
LIN {X 89.433,Y -29.727,Z -46.540,A -90.000,B 90.000,C 0.000} C_DIS
LIN {X 89.582,Y -29.705,Z -46.349,A -90.000,B 90.000,C 0.000} C_DIS
LIN {X 89.732,Y -29.691,Z -46.162,A -90.000,B 90.000,C 0.000} C_DIS
LIN {X 90.041,Y -29.658,Z -45.798,A -90.000,B 90.000,C 0.000} C_DIS
LIN {X 90.091,Y -29.652,Z -45.740,A -90.000,B 90.000,C 0.000} C_DIS
LIN {X 90.624,Y -29.580,Z -45.173,A -90.000,B 90.000,C 0.000} C_DIS
LIN {X 91.033,Y -29.544,Z -44.749,A -90.000,B 90.000,C 0.000} C_DIS
LIN {X 91.481,Y -29.506,Z -44.320,A -90.000,B 90.000,C 0.000} C_DIS
LIN {X 91.688,Y -29.492,Z -44.122,A -90.000,B 90.000,C 0.000} C_DIS
LIN {X 92.055,Y -29.466,Z -43.798,A -90.000,B 90.000,C 0.000} C_DIS
LIN {X 92.680,Y -29.419,Z -43.291,A -90.000,B 90.000,C 0.000} C_DIS
LIN {X 93.082,Y -29.400,Z -42.967,A -90.000,B 90.000,C 0.000} C_DIS
LIN {X 93.527,Y -29.381,Z -42.634,A -90.000,B 90.000,C 0.000} C_DIS
LIN {X 93.778,Y -29.370,Z -42.450,A -90.000,B 90.000,C 0.000} C_DIS
LIN {X 94.225,Y -29.352,Z -42.151,A -90.000,B 90.000,C 0.000} C_DIS
LIN {X 94.617,Y -29.341,Z -41.891,A -90.000,B 90.000,C 0.000} C_DIS
LIN {X 94.843,Y -29.334,Z -41.746,A -90.000,B 90.000,C 0.000} C_DIS
LIN {X 95.423,Y -29.323,Z -41.379,A -90.000,B 90.000,C 0.000} C_DIS
LIN {X 95.904,Y -29.317,Z -41.098,A -90.000,B 90.000,C 0.000} C_DIS
LIN {X 96.472,Y -29.312,Z -40.774,A -90.000,B 90.000,C 0.000} C_DIS
LIN {X 97.388,Y -29.309,Z -40.253,A -90.000,B 90.000,C 0.000} C_DIS
LIN {X 98.805,Y -29.308,Z -39.523,A -90.000,B 90.000,C 0.000} C_DIS
LIN {X 100.115,Y -29.305,Z -38.843,A -90.000,B 90.000,C 0.000} C_DIS
LIN {X 100.938,Y -29.298,Z -38.409,A -90.000,B 90.000,C 0.000} C_DIS
LIN {X 101.272,Y -29.292,Z -38.229,A -90.000,B 90.000,C 0.000} C_DIS
LIN {X 101.475,Y -29.286,Z -38.118,A -90.000,B 90.000,C 0.000} C_DIS
LIN {X 101.578,Y -29.279,Z -38.060,A -90.000,B 90.000,C 0.000} C_DIS
LIN {X 101.617,Y -29.273,Z -38.040,A -90.000,B 90.000,C 0.000} C_DIS
LIN {X 101.623,Y -29.271,Z -38.039,A -90.000,B 90.000,C 0.000} C_DIS
LIN {X 101.627,Y -29.266,Z -38.044,A -90.000,B 90.000,C 0.000} C_DIS
LIN {X 101.635,Y -29.264,Z -38.046,A -90.000,B 90.000,C 0.000} C_DIS
LIN {X 101.651,Y -29.263,Z -38.046,A -90.000,B 90.000,C 0.000} C_DIS
LIN {X 101.728,Y -29.262,Z -38.030,A -90.000,B 90.000,C 0.000} C_DIS
LIN {X 101.797,Y -29.262,Z -38.009,A -90.000,B 90.000,C 0.000} C_DIS
LIN {X 102.016,Y -29.264,Z -37.935,A -90.000,B 90.000,C 0.000} C_DIS
LIN {X 102.372,Y -29.270,Z -37.802,A -90.000,B 90.000,C 0.000} C_DIS
LIN {X 102.899,Y -29.279,Z -37.594,A -90.000,B 90.000,C 0.000} C_DIS
LIN {X 103.237,Y -29.284,Z -37.457,A -90.000,B 90.000,C 0.000} C_DIS
LIN {X 104.599,Y -29.308,Z -36.891,A -90.000,B 90.000,C 0.000} C_DIS
LIN {X 105.075,Y -29.317,Z -36.690,A -90.000,B 90.000,C 0.000} C_DIS
LIN {X 105.369,Y -29.308,Z -36.566,A -90.000,B 90.000,C 0.000} C_DIS
LIN {X 105.369,Y -60.000,Z -36.566,A -90.000,B 90.000,C 0.000} C_DIS
LIN {X 84.100,Y -60.000,Z -54.567,A -90.000,B 90.000,C 0.000} C_DIS
LIN {X 84.100,Y -29.308,Z -54.567,A -90.000,B 90.000,C 0.000} C_DIS
LIN {X 84.447,Y -29.442,Z -54.107,A -90.000,B 90.000,C 0.000} C_DIS
LIN {X 84.533,Y -29.476,Z -53.995,A -90.000,B 90.000,C 0.000} C_DIS
LIN {X 84.571,Y -29.454,Z -53.857,A -90.000,B 90.000,C 0.000} C_DIS
LIN {X 84.652,Y -29.405,Z -53.586,A -90.000,B 90.000,C 0.000} C_DIS
LIN {X 84.730,Y -29.308,Z -53.217,A -90.000,B 90.000,C 0.000} C_DIS
LIN {X 84.730,Y -60.000,Z -53.217,A -90.000,B 90.000,C 0.000} C_DIS
LIN {X 105.791,Y -60.000,Z -75.722,A -90.000,B 90.000,C 0.000} C_DIS
LIN {X 105.791,Y -29.308,Z -75.722,A -90.000,B 90.000,C 0.000} C_DIS
LIN {X 105.411,Y -29.308,Z -76.516,A -90.000,B 90.000,C 0.000} C_DIS
LIN {X 105.399,Y -29.308,Z -76.539,A -90.000,B 90.000,C 0.000} C_DIS
LIN {X 105.353,Y -29.308,Z -76.624,A -90.000,B 90.000,C 0.000} C_DIS
LIN {X 105.168,Y -29.308,Z -76.983,A -90.000,B 90.000,C 0.000} C_DIS
LIN {X 104.922,Y -29.307,Z -77.443,A -90.000,B 90.000,C 0.000} C_DIS
LIN {X 104.819,Y -29.304,Z -77.654,A -90.000,B 90.000,C 0.000} C_DIS
LIN {X 104.799,Y -29.302,Z -77.707,A -90.000,B 90.000,C 0.000} C_DIS
LIN {X 104.798,Y -29.301,Z -77.713,A -90.000,B 90.000,C 0.000} C_DIS
LIN {X 104.801,Y -29.299,Z -77.720,A -90.000,B 90.000,C 0.000} C_DIS
LIN {X 104.773,Y -29.299,Z -77.776,A -90.000,B 90.000,C 0.000} C_DIS
LIN {X 104.197,Y -29.308,Z -78.782,A -90.000,B 90.000,C 0.000} C_DIS
LIN {X 104.093,Y -29.310,Z -78.964,A -90.000,B 90.000,C 0.000} C_DIS
LIN {X 103.987,Y -29.308,Z -79.149,A -90.000,B 90.000,C 0.000} C_DIS
LIN {X 103.987,Y -60.000,Z -79.149,A -90.000,B 90.000,C 0.000} C_DIS
LIN {X -25.435,Y -60.000,Z -59.019,A -90.000,B 90.000,C 0.000} C_DIS
LIN {X -25.435,Y -29.308,Z -59.019,A -90.000,B 90.000,C 0.000} C_DIS
LIN {X -25.318,Y -29.314,Z -59.040,A -90.000,B 90.000,C 0.000} C_DIS
LIN {X -24.855,Y -29.356,Z -59.112,A -90.000,B 90.000,C 0.000} C_DIS
LIN {X -24.743,Y -29.308,Z -59.029,A -90.000,B 90.000,C 0.000} C_DIS
LIN {X -24.743,Y -60.000,Z -59.029,A -90.000,B 90.000,C 0.000} C_DIS
LIN {X -60.245,Y -60.000,Z -86.406,A -90.000,B 90.000,C 0.000} C_DIS
LIN {X -60.245,Y -29.308,Z -86.406,A -90.000,B 90.000,C 0.000} C_DIS
LIN {X -60.476,Y -29.386,Z -85.949,A -90.000,B 90.000,C 0.000} C_DIS
LIN {X -60.969,Y -29.507,Z -85.064,A -90.000,B 90.000,C 0.000} C_DIS
LIN {X -61.117,Y -29.536,Z -84.790,A -90.000,B 90.000,C 0.000} C_DIS
LIN {X -61.503,Y -29.612,Z -84.088,A -90.000,B 90.000,C 0.000} C_DIS
LIN {X -61.609,Y -29.631,Z -83.891,A -90.000,B 90.000,C 0.000} C_DIS
LIN {X -61.656,Y -29.639,Z -83.795,A -90.000,B 90.000,C 0.000} C_DIS
LIN {X -61.696,Y -29.647,Z -83.709,A -90.000,B 90.000,C 0.000} C_DIS
LIN {X -61.785,Y -29.670,Z -83.501,A -90.000,B 90.000,C 0.000} C_DIS
LIN {X -61.967,Y -29.722,Z -83.061,A -90.000,B 90.000,C 0.000} C_DIS
LIN {X -62.117,Y -29.776,Z -82.698,A -90.000,B 90.000,C 0.000} C_DIS
LIN {X -62.458,Y -29.864,Z -81.977,A -90.000,B 90.000,C 0.000} C_DIS
LIN {X -62.540,Y -29.889,Z -81.810,A -90.000,B 90.000,C 0.000} C_DIS
LIN {X -62.957,Y -29.989,Z -80.941,A -90.000,B 90.000,C 0.000} C_DIS
LIN {X -62.980,Y -29.996,Z -80.890,A -90.000,B 90.000,C 0.000} C_DIS
LIN {X -63.125,Y -30.020,Z -80.544,A -90.000,B 90.000,C 0.000} C_DIS
LIN {X -63.312,Y -30.056,Z -80.074,A -90.000,B 90.000,C 0.000} C_DIS
LIN {X -63.389,Y -30.070,Z -79.879,A -90.000,B 90.000,C 0.000} C_DIS
LIN {X -63.558,Y -30.099,Z -79.504,A -90.000,B 90.000,C 0.000} C_DIS
LIN {X -63.658,Y -30.116,Z -79.286,A -90.000,B 90.000,C 0.000} C_DIS
LIN {X -63.738,Y -30.128,Z -79.100,A -90.000,B 90.000,C 0.000} C_DIS
LIN {X -63.785,Y -30.141,Z -78.988,A -90.000,B 90.000,C 0.000} C_DIS
LIN {X -64.069,Y -30.208,Z -78.260,A -90.000,B 90.000,C 0.000} C_DIS
LIN {X -64.147,Y -30.219,Z -78.049,A -90.000,B 90.000,C 0.000} C_DIS
LIN {X -64.342,Y -30.238,Z -77.496,A -90.000,B 90.000,C 0.000} C_DIS
LIN {X -64.479,Y -30.266,Z -77.112,A -90.000,B 90.000,C 0.000} C_DIS
LIN {X -64.598,Y -30.296,Z -76.743,A -90.000,B 90.000,C 0.000} C_DIS
LIN {X -64.679,Y -30.313,Z -76.467,A -90.000,B 90.000,C 0.000} C_DIS
LIN {X -64.845,Y -30.347,Z -75.884,A -90.000,B 90.000,C 0.000} C_DIS
LIN {X -64.928,Y -30.363,Z -75.587,A -90.000,B 90.000,C 0.000} C_DIS
LIN {X -65.166,Y -30.400,Z -74.801,A -90.000,B 90.000,C 0.000} C_DIS
LIN {X -65.391,Y -30.424,Z -74.139,A -90.000,B 90.000,C 0.000} C_DIS
LIN {X -65.541,Y -30.424,Z -73.773,A -90.000,B 90.000,C 0.000} C_DIS
LIN {X -65.582,Y -30.424,Z -73.668,A -90.000,B 90.000,C 0.000} C_DIS
LIN {X -65.706,Y -30.431,Z -73.323,A -90.000,B 90.000,C 0.000} C_DIS
LIN {X -66.010,Y -30.426,Z -72.678,A -90.000,B 90.000,C 0.000} C_DIS
LIN {X -66.059,Y -30.426,Z -72.567,A -90.000,B 90.000,C 0.000} C_DIS
LIN {X -66.099,Y -30.429,Z -72.463,A -90.000,B 90.000,C 0.000} C_DIS
LIN {X -66.363,Y -30.428,Z -71.965,A -90.000,B 90.000,C 0.000} C_DIS
LIN {X -66.493,Y -30.424,Z -71.746,A -90.000,B 90.000,C 0.000} C_DIS
LIN {X -66.736,Y -30.422,Z -71.318,A -90.000,B 90.000,C 0.000} C_DIS
LIN {X -66.924,Y -30.413,Z -71.070,A -90.000,B 90.000,C 0.000} C_DIS
LIN {X -67.348,Y -30.412,Z -70.514,A -90.000,B 90.000,C 0.000} C_DIS
LIN {X -67.491,Y -30.409,Z -70.320,A -90.000,B 90.000,C 0.000} C_DIS
LIN {X -68.041,Y -30.435,Z -69.506,A -90.000,B 90.000,C 0.000} C_DIS
LIN {X -68.477,Y -30.457,Z -68.893,A -90.000,B 90.000,C 0.000} C_DIS
LIN {X -68.662,Y -30.474,Z -68.637,A -90.000,B 90.000,C 0.000} C_DIS
LIN {X -68.812,Y -30.483,Z -68.426,A -90.000,B 90.000,C 0.000} C_DIS
LIN {X -68.960,Y -30.495,Z -68.201,A -90.000,B 90.000,C 0.000} C_DIS
LIN {X -69.046,Y -30.508,Z -68.056,A -90.000,B 90.000,C 0.000} C_DIS
LIN {X -69.107,Y -30.520,Z -67.945,A -90.000,B 90.000,C 0.000} C_DIS
LIN {X -69.220,Y -30.546,Z -67.711,A -90.000,B 90.000,C 0.000} C_DIS
LIN {X -69.389,Y -30.595,Z -67.310,A -90.000,B 90.000,C 0.000} C_DIS
LIN {X -69.510,Y -30.635,Z -66.994,A -90.000,B 90.000,C 0.000} C_DIS
LIN {X -69.550,Y -30.648,Z -66.884,A -90.000,B 90.000,C 0.000} C_DIS
LIN {X -69.575,Y -30.657,Z -66.801,A -90.000,B 90.000,C 0.000} C_DIS
LIN {X -69.655,Y -30.690,Z -66.508,A -90.000,B 90.000,C 0.000} C_DIS
LIN {X -69.744,Y -30.738,Z -66.107,A -90.000,B 90.000,C 0.000} C_DIS
LIN {X -69.801,Y -30.764,Z -65.841,A -90.000,B 90.000,C 0.000} C_DIS
LIN {X -69.833,Y -30.788,Z -65.632,A -90.000,B 90.000,C 0.000} C_DIS
LIN {X -69.860,Y -30.803,Z -65.432,A -90.000,B 90.000,C 0.000} C_DIS
LIN {X -69.882,Y -30.824,Z -65.125,A -90.000,B 90.000,C 0.000} C_DIS
LIN {X -69.886,Y -30.833,Z -65.000,A -90.000,B 90.000,C 0.000} C_DIS
LIN {X -69.886,Y -30.845,Z -64.839,A -90.000,B 90.000,C 0.000} C_DIS
LIN {X -69.883,Y -30.854,Z -64.720,A -90.000,B 90.000,C 0.000} C_DIS
LIN {X -69.871,Y -30.861,Z -64.554,A -90.000,B 90.000,C 0.000} C_DIS
LIN {X -69.854,Y -30.863,Z -64.409,A -90.000,B 90.000,C 0.000} C_DIS
LIN {X -69.818,Y -30.862,Z -64.197,A -90.000,B 90.000,C 0.000} C_DIS
LIN {X -69.791,Y -30.860,Z -64.064,A -90.000,B 90.000,C 0.000} C_DIS
LIN {X -69.739,Y -30.858,Z -63.834,A -90.000,B 90.000,C 0.000} C_DIS
LIN {X -69.701,Y -30.857,Z -63.690,A -90.000,B 90.000,C 0.000} C_DIS
LIN {X -69.652,Y -30.856,Z -63.528,A -90.000,B 90.000,C 0.000} C_DIS
LIN {X -69.596,Y -30.854,Z -63.376,A -90.000,B 90.000,C 0.000} C_DIS
LIN {X -69.562,Y -30.852,Z -63.297,A -90.000,B 90.000,C 0.000} C_DIS
LIN {X -69.505,Y -30.845,Z -63.168,A -90.000,B 90.000,C 0.000} C_DIS
LIN {X -69.455,Y -30.832,Z -63.058,A -90.000,B 90.000,C 0.000} C_DIS
LIN {X -69.398,Y -30.817,Z -62.937,A -90.000,B 90.000,C 0.000} C_DIS
LIN {X -69.100,Y -30.749,Z -62.404,A -90.000,B 90.000,C 0.000} C_DIS
LIN {X -69.008,Y -30.730,Z -62.251,A -90.000,B 90.000,C 0.000} C_DIS
LIN {X -68.931,Y -30.715,Z -62.135,A -90.000,B 90.000,C 0.000} C_DIS
LIN {X -68.867,Y -30.705,Z -62.044,A -90.000,B 90.000,C 0.000} C_DIS
LIN {X -68.813,Y -30.696,Z -61.971,A -90.000,B 90.000,C 0.000} C_DIS
LIN {X -68.715,Y -30.682,Z -61.849,A -90.000,B 90.000,C 0.000} C_DIS
LIN {X -68.634,Y -30.662,Z -61.754,A -90.000,B 90.000,C 0.000} C_DIS
LIN {X -68.210,Y -30.561,Z -61.276,A -90.000,B 90.000,C 0.000} C_DIS
LIN {X -68.149,Y -30.547,Z -61.210,A -90.000,B 90.000,C 0.000} C_DIS
LIN {X -67.971,Y -30.512,Z -61.028,A -90.000,B 90.000,C 0.000} C_DIS
LIN {X -67.811,Y -30.480,Z -60.876,A -90.000,B 90.000,C 0.000} C_DIS
LIN {X -67.705,Y -30.460,Z -60.783,A -90.000,B 90.000,C 0.000} C_DIS
LIN {X -67.616,Y -30.444,Z -60.709,A -90.000,B 90.000,C 0.000} C_DIS
LIN {X -67.384,Y -30.408,Z -60.535,A -90.000,B 90.000,C 0.000} C_DIS
LIN {X -67.255,Y -30.389,Z -60.450,A -90.000,B 90.000,C 0.000} C_DIS
LIN {X -67.127,Y -30.372,Z -60.372,A -90.000,B 90.000,C 0.000} C_DIS
LIN {X -67.027,Y -30.360,Z -60.314,A -90.000,B 90.000,C 0.000} C_DIS
LIN {X -66.800,Y -30.335,Z -60.191,A -90.000,B 90.000,C 0.000} C_DIS
LIN {X -66.681,Y -30.323,Z -60.131,A -90.000,B 90.000,C 0.000} C_DIS
LIN {X -66.236,Y -30.282,Z -59.917,A -90.000,B 90.000,C 0.000} C_DIS
LIN {X -65.984,Y -30.260,Z -59.800,A -90.000,B 90.000,C 0.000} C_DIS
LIN {X -65.745,Y -30.241,Z -59.696,A -90.000,B 90.000,C 0.000} C_DIS
LIN {X -65.501,Y -30.226,Z -59.602,A -90.000,B 90.000,C 0.000} C_DIS
LIN {X -65.417,Y -30.222,Z -59.572,A -90.000,B 90.000,C 0.000} C_DIS
LIN {X -64.705,Y -30.190,Z -59.341,A -90.000,B 90.000,C 0.000} C_DIS
LIN {X -63.703,Y -30.140,Z -59.006,A -90.000,B 90.000,C 0.000} C_DIS
LIN {X -63.245,Y -30.124,Z -58.851,A -90.000,B 90.000,C 0.000} C_DIS
LIN {X -63.141,Y -30.121,Z -58.819,A -90.000,B 90.000,C 0.000} C_DIS
LIN {X -62.935,Y -30.117,Z -58.761,A -90.000,B 90.000,C 0.000} C_DIS
LIN {X -62.761,Y -30.116,Z -58.719,A -90.000,B 90.000,C 0.000} C_DIS
LIN {X -61.998,Y -30.115,Z -58.547,A -90.000,B 90.000,C 0.000} C_DIS
LIN {X -61.360,Y -30.120,Z -58.416,A -90.000,B 90.000,C 0.000} C_DIS
LIN {X -61.045,Y -30.126,Z -58.352,A -90.000,B 90.000,C 0.000} C_DIS
LIN {X -60.753,Y -30.129,Z -58.299,A -90.000,B 90.000,C 0.000} C_DIS
LIN {X -58.944,Y -30.146,Z -57.971,A -90.000,B 90.000,C 0.000} C_DIS
LIN {X -58.179,Y -30.156,Z -57.841,A -90.000,B 90.000,C 0.000} C_DIS
LIN {X -57.741,Y -30.164,Z -57.766,A -90.000,B 90.000,C 0.000} C_DIS
LIN {X -56.817,Y -30.174,Z -57.612,A -90.000,B 90.000,C 0.000} C_DIS
LIN {X -54.566,Y -30.204,Z -57.295,A -90.000,B 90.000,C 0.000} C_DIS
LIN {X -53.759,Y -30.212,Z -57.181,A -90.000,B 90.000,C 0.000} C_DIS
LIN {X -52.829,Y -30.214,Z -57.045,A -90.000,B 90.000,C 0.000} C_DIS
LIN {X -51.830,Y -30.214,Z -56.894,A -90.000,B 90.000,C 0.000} C_DIS
LIN {X -51.067,Y -30.197,Z -56.787,A -90.000,B 90.000,C 0.000} C_DIS
LIN {X -50.180,Y -30.172,Z -56.664,A -90.000,B 90.000,C 0.000} C_DIS
LIN {X -49.770,Y -30.159,Z -56.606,A -90.000,B 90.000,C 0.000} C_DIS
LIN {X -49.570,Y -30.152,Z -56.575,A -90.000,B 90.000,C 0.000} C_DIS
LIN {X -48.724,Y -30.089,Z -56.454,A -90.000,B 90.000,C 0.000} C_DIS
LIN {X -48.521,Y -30.078,Z -56.423,A -90.000,B 90.000,C 0.000} C_DIS
LIN {X -47.719,Y -30.011,Z -56.295,A -90.000,B 90.000,C 0.000} C_DIS
LIN {X -47.499,Y -29.986,Z -56.263,A -90.000,B 90.000,C 0.000} C_DIS
LIN {X -47.255,Y -29.952,Z -56.232,A -90.000,B 90.000,C 0.000} C_DIS
LIN {X -46.661,Y -29.878,Z -56.171,A -90.000,B 90.000,C 0.000} C_DIS
LIN {X -46.399,Y -29.843,Z -56.145,A -90.000,B 90.000,C 0.000} C_DIS
LIN {X -45.541,Y -29.736,Z -56.061,A -90.000,B 90.000,C 0.000} C_DIS
LIN {X -45.135,Y -29.665,Z -56.032,A -90.000,B 90.000,C 0.000} C_DIS
LIN {X -44.600,Y -29.583,Z -56.011,A -90.000,B 90.000,C 0.000} C_DIS
LIN {X -44.202,Y -29.520,Z -56.012,A -90.000,B 90.000,C 0.000} C_DIS
LIN {X -43.159,Y -29.349,Z -56.017,A -90.000,B 90.000,C 0.000} C_DIS
LIN {X -42.926,Y -29.308,Z -56.022,A -90.000,B 90.000,C 0.000} C_DIS
LIN {X -42.926,Y -60.000,Z -56.022,A -90.000,B 90.000,C 0.000} C_DIS
LIN {X -65.501,Y -60.000,Z -79.588,A -90.000,B 90.000,C 0.000} C_DIS
LIN {X -65.501,Y -29.308,Z -79.588,A -90.000,B 90.000,C 0.000} C_DIS
LIN {X -65.847,Y -29.426,Z -78.751,A -90.000,B 90.000,C 0.000} C_DIS
LIN {X -65.900,Y -29.437,Z -78.611,A -90.000,B 90.000,C 0.000} C_DIS
LIN {X -65.998,Y -29.469,Z -78.363,A -90.000,B 90.000,C 0.000} C_DIS
LIN {X -66.173,Y -29.522,Z -77.908,A -90.000,B 90.000,C 0.000} C_DIS
LIN {X -66.276,Y -29.556,Z -77.631,A -90.000,B 90.000,C 0.000} C_DIS
LIN {X -66.422,Y -29.613,Z -77.200,A -90.000,B 90.000,C 0.000} C_DIS
LIN {X -66.668,Y -29.698,Z -76.391,A -90.000,B 90.000,C 0.000} C_DIS
LIN {X -66.756,Y -29.729,Z -76.093,A -90.000,B 90.000,C 0.000} C_DIS
LIN {X -66.990,Y -29.799,Z -75.361,A -90.000,B 90.000,C 0.000} C_DIS
LIN {X -67.185,Y -29.837,Z -74.803,A -90.000,B 90.000,C 0.000} C_DIS
LIN {X -67.334,Y -29.854,Z -74.452,A -90.000,B 90.000,C 0.000} C_DIS
LIN {X -67.391,Y -29.863,Z -74.308,A -90.000,B 90.000,C 0.000} C_DIS
LIN {X -67.485,Y -29.879,Z -74.058,A -90.000,B 90.000,C 0.000} C_DIS
LIN {X -67.679,Y -29.897,Z -73.660,A -90.000,B 90.000,C 0.000} C_DIS
LIN {X -67.780,Y -29.902,Z -73.447,A -90.000,B 90.000,C 0.000} C_DIS
LIN {X -67.859,Y -29.908,Z -73.267,A -90.000,B 90.000,C 0.000} C_DIS
LIN {X -68.047,Y -29.911,Z -72.913,A -90.000,B 90.000,C 0.000} C_DIS
LIN {X -68.211,Y -29.909,Z -72.634,A -90.000,B 90.000,C 0.000} C_DIS
LIN {X -68.350,Y -29.911,Z -72.392,A -90.000,B 90.000,C 0.000} C_DIS
LIN {X -68.486,Y -29.906,Z -72.212,A -90.000,B 90.000,C 0.000} C_DIS
LIN {X -68.869,Y -29.900,Z -71.708,A -90.000,B 90.000,C 0.000} C_DIS
LIN {X -69.046,Y -29.904,Z -71.471,A -90.000,B 90.000,C 0.000} C_DIS
LIN {X -69.123,Y -29.906,Z -71.362,A -90.000,B 90.000,C 0.000} C_DIS
LIN {X -69.507,Y -29.922,Z -70.792,A -90.000,B 90.000,C 0.000} C_DIS
LIN {X -69.652,Y -29.925,Z -70.577,A -90.000,B 90.000,C 0.000} C_DIS
LIN {X -69.819,Y -29.927,Z -70.339,A -90.000,B 90.000,C 0.000} C_DIS
LIN {X -69.963,Y -29.938,Z -70.138,A -90.000,B 90.000,C 0.000} C_DIS
LIN {X -70.153,Y -29.952,Z -69.874,A -90.000,B 90.000,C 0.000} C_DIS
LIN {X -70.331,Y -29.970,Z -69.628,A -90.000,B 90.000,C 0.000} C_DIS
LIN {X -70.443,Y -29.980,Z -69.469,A -90.000,B 90.000,C 0.000} C_DIS
LIN {X -70.625,Y -29.999,Z -69.192,A -90.000,B 90.000,C 0.000} C_DIS
LIN {X -70.728,Y -30.018,Z -69.019,A -90.000,B 90.000,C 0.000} C_DIS
LIN {X -70.847,Y -30.044,Z -68.808,A -90.000,B 90.000,C 0.000} C_DIS
LIN {X -70.990,Y -30.076,Z -68.515,A -90.000,B 90.000,C 0.000} C_DIS
LIN {X -71.028,Y -30.085,Z -68.432,A -90.000,B 90.000,C 0.000} C_DIS
LIN {X -71.231,Y -30.155,Z -67.955,A -90.000,B 90.000,C 0.000} C_DIS
LIN {X -71.309,Y -30.181,Z -67.751,A -90.000,B 90.000,C 0.000} C_DIS
LIN {X -71.419,Y -30.227,Z -67.457,A -90.000,B 90.000,C 0.000} C_DIS
LIN {X -71.477,Y -30.257,Z -67.275,A -90.000,B 90.000,C 0.000} C_DIS
LIN {X -71.548,Y -30.300,Z -67.024,A -90.000,B 90.000,C 0.000} C_DIS
LIN {X -71.585,Y -30.325,Z -66.884,A -90.000,B 90.000,C 0.000} C_DIS
LIN {X -71.676,Y -30.394,Z -66.496,A -90.000,B 90.000,C 0.000} C_DIS
LIN {X -71.737,Y -30.434,Z -66.222,A -90.000,B 90.000,C 0.000} C_DIS
LIN {X -71.765,Y -30.457,Z -66.069,A -90.000,B 90.000,C 0.000} C_DIS
LIN {X -71.812,Y -30.505,Z -65.758,A -90.000,B 90.000,C 0.000} C_DIS
LIN {X -71.830,Y -30.519,Z -65.631,A -90.000,B 90.000,C 0.000} C_DIS
LIN {X -71.858,Y -30.563,Z -65.297,A -90.000,B 90.000,C 0.000} C_DIS
LIN {X -71.870,Y -30.586,Z -65.050,A -90.000,B 90.000,C 0.000} C_DIS
LIN {X -71.872,Y -30.613,Z -64.767,A -90.000,B 90.000,C 0.000} C_DIS
LIN {X -71.867,Y -30.632,Z -64.600,A -90.000,B 90.000,C 0.000} C_DIS
LIN {X -71.858,Y -30.642,Z -64.471,A -90.000,B 90.000,C 0.000} C_DIS
LIN {X -71.845,Y -30.650,Z -64.312,A -90.000,B 90.000,C 0.000} C_DIS
LIN {X -71.825,Y -30.653,Z -64.137,A -90.000,B 90.000,C 0.000} C_DIS
LIN {X -71.770,Y -30.655,Z -63.816,A -90.000,B 90.000,C 0.000} C_DIS
LIN {X -71.731,Y -30.656,Z -63.620,A -90.000,B 90.000,C 0.000} C_DIS
LIN {X -71.663,Y -30.657,Z -63.328,A -90.000,B 90.000,C 0.000} C_DIS
LIN {X -71.631,Y -30.655,Z -63.207,A -90.000,B 90.000,C 0.000} C_DIS
LIN {X -71.588,Y -30.651,Z -63.059,A -90.000,B 90.000,C 0.000} C_DIS
LIN {X -71.548,Y -30.643,Z -62.931,A -90.000,B 90.000,C 0.000} C_DIS
LIN {X -71.497,Y -30.626,Z -62.788,A -90.000,B 90.000,C 0.000} C_DIS
LIN {X -71.457,Y -30.613,Z -62.683,A -90.000,B 90.000,C 0.000} C_DIS
LIN {X -71.403,Y -30.598,Z -62.558,A -90.000,B 90.000,C 0.000} C_DIS
LIN {X -71.256,Y -30.561,Z -62.230,A -90.000,B 90.000,C 0.000} C_DIS
LIN {X -71.182,Y -30.543,Z -62.077,A -90.000,B 90.000,C 0.000} C_DIS
LIN {X -71.099,Y -30.522,Z -61.925,A -90.000,B 90.000,C 0.000} C_DIS
LIN {X -70.943,Y -30.484,Z -61.646,A -90.000,B 90.000,C 0.000} C_DIS
LIN {X -70.808,Y -30.432,Z -61.414,A -90.000,B 90.000,C 0.000} C_DIS
LIN {X -70.673,Y -30.384,Z -61.199,A -90.000,B 90.000,C 0.000} C_DIS
LIN {X -70.562,Y -30.349,Z -61.037,A -90.000,B 90.000,C 0.000} C_DIS
LIN {X -70.380,Y -30.300,Z -60.792,A -90.000,B 90.000,C 0.000} C_DIS
LIN {X -70.325,Y -30.286,Z -60.726,A -90.000,B 90.000,C 0.000} C_DIS
LIN {X -70.140,Y -30.232,Z -60.509,A -90.000,B 90.000,C 0.000} C_DIS
LIN {X -69.681,Y -30.104,Z -60.000,A -90.000,B 90.000,C 0.000} C_DIS
LIN {X -69.582,Y -30.078,Z -59.896,A -90.000,B 90.000,C 0.000} C_DIS
LIN {X -69.358,Y -30.022,Z -59.674,A -90.000,B 90.000,C 0.000} C_DIS
LIN {X -69.140,Y -29.972,Z -59.471,A -90.000,B 90.000,C 0.000} C_DIS
LIN {X -68.915,Y -29.925,Z -59.279,A -90.000,B 90.000,C 0.000} C_DIS
LIN {X -68.823,Y -29.908,Z -59.207,A -90.000,B 90.000,C 0.000} C_DIS
LIN {X -68.616,Y -29.871,Z -59.054,A -90.000,B 90.000,C 0.000} C_DIS
LIN {X -68.492,Y -29.850,Z -58.966,A -90.000,B 90.000,C 0.000} C_DIS
LIN {X -68.316,Y -29.824,Z -58.852,A -90.000,B 90.000,C 0.000} C_DIS
LIN {X -68.138,Y -29.800,Z -58.743,A -90.000,B 90.000,C 0.000} C_DIS
LIN {X -67.983,Y -29.781,Z -58.655,A -90.000,B 90.000,C 0.000} C_DIS
LIN {X -67.678,Y -29.747,Z -58.493,A -90.000,B 90.000,C 0.000} C_DIS
LIN {X -67.556,Y -29.736,Z -58.431,A -90.000,B 90.000,C 0.000} C_DIS
LIN {X -67.133,Y -29.705,Z -58.225,A -90.000,B 90.000,C 0.000} C_DIS
LIN {X -66.788,Y -29.681,Z -58.063,A -90.000,B 90.000,C 0.000} C_DIS
LIN {X -66.549,Y -29.669,Z -57.957,A -90.000,B 90.000,C 0.000} C_DIS
LIN {X -66.463,Y -29.666,Z -57.920,A -90.000,B 90.000,C 0.000} C_DIS
LIN {X -66.116,Y -29.654,Z -57.786,A -90.000,B 90.000,C 0.000} C_DIS
LIN {X -65.648,Y -29.645,Z -57.629,A -90.000,B 90.000,C 0.000} C_DIS
LIN {X -65.330,Y -29.644,Z -57.521,A -90.000,B 90.000,C 0.000} C_DIS
LIN {X -64.338,Y -29.639,Z -57.177,A -90.000,B 90.000,C 0.000} C_DIS
LIN {X -64.036,Y -29.642,Z -57.071,A -90.000,B 90.000,C 0.000} C_DIS
LIN {X -63.831,Y -29.641,Z -57.001,A -90.000,B 90.000,C 0.000} C_DIS
LIN {X -63.676,Y -29.640,Z -56.953,A -90.000,B 90.000,C 0.000} C_DIS
LIN {X -63.397,Y -29.642,Z -56.874,A -90.000,B 90.000,C 0.000} C_DIS
LIN {X -63.190,Y -29.645,Z -56.823,A -90.000,B 90.000,C 0.000} C_DIS
LIN {X -62.975,Y -29.648,Z -56.774,A -90.000,B 90.000,C 0.000} C_DIS
LIN {X -62.384,Y -29.665,Z -56.637,A -90.000,B 90.000,C 0.000} C_DIS
LIN {X -61.390,Y -29.695,Z -56.429,A -90.000,B 90.000,C 0.000} C_DIS
LIN {X -60.796,Y -29.720,Z -56.318,A -90.000,B 90.000,C 0.000} C_DIS
LIN {X -59.627,Y -29.743,Z -56.103,A -90.000,B 90.000,C 0.000} C_DIS
LIN {X -59.289,Y -29.748,Z -56.042,A -90.000,B 90.000,C 0.000} C_DIS
LIN {X -57.787,Y -29.773,Z -55.786,A -90.000,B 90.000,C 0.000} C_DIS
LIN {X -57.385,Y -29.777,Z -55.718,A -90.000,B 90.000,C 0.000} C_DIS
LIN {X -57.137,Y -29.777,Z -55.677,A -90.000,B 90.000,C 0.000} C_DIS
LIN {X -55.206,Y -29.750,Z -55.417,A -90.000,B 90.000,C 0.000} C_DIS
LIN {X -54.540,Y -29.734,Z -55.328,A -90.000,B 90.000,C 0.000} C_DIS
LIN {X -53.923,Y -29.716,Z -55.247,A -90.000,B 90.000,C 0.000} C_DIS
LIN {X -53.104,Y -29.659,Z -55.144,A -90.000,B 90.000,C 0.000} C_DIS
LIN {X -52.397,Y -29.610,Z -55.052,A -90.000,B 90.000,C 0.000} C_DIS
LIN {X -51.317,Y -29.527,Z -54.919,A -90.000,B 90.000,C 0.000} C_DIS
LIN {X -51.150,Y -29.512,Z -54.899,A -90.000,B 90.000,C 0.000} C_DIS
LIN {X -50.066,Y -29.377,Z -54.789,A -90.000,B 90.000,C 0.000} C_DIS
LIN {X -49.587,Y -29.308,Z -54.736,A -90.000,B 90.000,C 0.000} C_DIS
LIN {X -49.587,Y -60.000,Z -54.736,A -90.000,B 90.000,C 0.000} C_DIS
LIN {X -71.239,Y -60.000,Z -71.627,A -90.000,B 90.000,C 0.000} C_DIS
LIN {X -71.239,Y -29.308,Z -71.627,A -90.000,B 90.000,C 0.000} C_DIS
LIN {X -71.612,Y -29.349,Z -71.115,A -90.000,B 90.000,C 0.000} C_DIS
LIN {X -71.828,Y -29.367,Z -70.815,A -90.000,B 90.000,C 0.000} C_DIS
LIN {X -72.060,Y -29.397,Z -70.491,A -90.000,B 90.000,C 0.000} C_DIS
LIN {X -72.222,Y -29.423,Z -70.250,A -90.000,B 90.000,C 0.000} C_DIS
LIN {X -72.279,Y -29.437,Z -70.166,A -90.000,B 90.000,C 0.000} C_DIS
LIN {X -72.432,Y -29.469,Z -69.911,A -90.000,B 90.000,C 0.000} C_DIS
LIN {X -72.566,Y -29.500,Z -69.674,A -90.000,B 90.000,C 0.000} C_DIS
LIN {X -72.708,Y -29.550,Z -69.399,A -90.000,B 90.000,C 0.000} C_DIS
LIN {X -72.802,Y -29.578,Z -69.205,A -90.000,B 90.000,C 0.000} C_DIS
LIN {X -72.859,Y -29.597,Z -69.075,A -90.000,B 90.000,C 0.000} C_DIS
LIN {X -73.043,Y -29.674,Z -68.650,A -90.000,B 90.000,C 0.000} C_DIS
LIN {X -73.198,Y -29.740,Z -68.254,A -90.000,B 90.000,C 0.000} C_DIS
LIN {X -73.278,Y -29.779,Z -68.045,A -90.000,B 90.000,C 0.000} C_DIS
LIN {X -73.376,Y -29.838,Z -67.742,A -90.000,B 90.000,C 0.000} C_DIS
LIN {X -73.471,Y -29.907,Z -67.412,A -90.000,B 90.000,C 0.000} C_DIS
LIN {X -73.510,Y -29.936,Z -67.264,A -90.000,B 90.000,C 0.000} C_DIS
LIN {X -73.604,Y -30.018,Z -66.869,A -90.000,B 90.000,C 0.000} C_DIS
LIN {X -73.683,Y -30.089,Z -66.525,A -90.000,B 90.000,C 0.000} C_DIS
LIN {X -73.712,Y -30.121,Z -66.379,A -90.000,B 90.000,C 0.000} C_DIS
LIN {X -73.751,Y -30.173,Z -66.149,A -90.000,B 90.000,C 0.000} C_DIS
LIN {X -73.796,Y -30.226,Z -65.853,A -90.000,B 90.000,C 0.000} C_DIS
LIN {X -73.807,Y -30.244,Z -65.760,A -90.000,B 90.000,C 0.000} C_DIS
LIN {X -73.830,Y -30.294,Z -65.508,A -90.000,B 90.000,C 0.000} C_DIS
LIN {X -73.843,Y -30.321,Z -65.326,A -90.000,B 90.000,C 0.000} C_DIS
LIN {X -73.857,Y -30.362,Z -65.062,A -90.000,B 90.000,C 0.000} C_DIS
LIN {X -73.860,Y -30.396,Z -64.781,A -90.000,B 90.000,C 0.000} C_DIS
LIN {X -73.856,Y -30.426,Z -64.552,A -90.000,B 90.000,C 0.000} C_DIS
LIN {X -73.849,Y -30.448,Z -64.392,A -90.000,B 90.000,C 0.000} C_DIS
LIN {X -73.843,Y -30.458,Z -64.302,A -90.000,B 90.000,C 0.000} C_DIS
LIN {X -73.825,Y -30.470,Z -64.092,A -90.000,B 90.000,C 0.000} C_DIS
LIN {X -73.796,Y -30.481,Z -63.849,A -90.000,B 90.000,C 0.000} C_DIS
LIN {X -73.756,Y -30.484,Z -63.608,A -90.000,B 90.000,C 0.000} C_DIS
LIN {X -73.718,Y -30.491,Z -63.391,A -90.000,B 90.000,C 0.000} C_DIS
LIN {X -73.673,Y -30.498,Z -63.168,A -90.000,B 90.000,C 0.000} C_DIS
LIN {X -73.641,Y -30.496,Z -63.031,A -90.000,B 90.000,C 0.000} C_DIS
LIN {X -73.590,Y -30.485,Z -62.820,A -90.000,B 90.000,C 0.000} C_DIS
LIN {X -73.532,Y -30.472,Z -62.611,A -90.000,B 90.000,C 0.000} C_DIS
LIN {X -73.452,Y -30.442,Z -62.352,A -90.000,B 90.000,C 0.000} C_DIS
LIN {X -73.365,Y -30.414,Z -62.108,A -90.000,B 90.000,C 0.000} C_DIS
LIN {X -73.312,Y -30.399,Z -61.968,A -90.000,B 90.000,C 0.000} C_DIS
LIN {X -73.270,Y -30.389,Z -61.868,A -90.000,B 90.000,C 0.000} C_DIS
LIN {X -73.180,Y -30.356,Z -61.665,A -90.000,B 90.000,C 0.000} C_DIS
LIN {X -73.056,Y -30.312,Z -61.396,A -90.000,B 90.000,C 0.000} C_DIS
LIN {X -72.963,Y -30.271,Z -61.209,A -90.000,B 90.000,C 0.000} C_DIS
LIN {X -72.868,Y -30.233,Z -61.037,A -90.000,B 90.000,C 0.000} C_DIS
LIN {X -72.580,Y -30.128,Z -60.534,A -90.000,B 90.000,C 0.000} C_DIS
LIN {X -72.510,Y -30.095,Z -60.418,A -90.000,B 90.000,C 0.000} C_DIS
LIN {X -72.331,Y -30.017,Z -60.143,A -90.000,B 90.000,C 0.000} C_DIS
LIN {X -72.172,Y -29.952,Z -59.918,A -90.000,B 90.000,C 0.000} C_DIS
LIN {X -71.999,Y -29.892,Z -59.692,A -90.000,B 90.000,C 0.000} C_DIS
LIN {X -71.900,Y -29.860,Z -59.569,A -90.000,B 90.000,C 0.000} C_DIS
LIN {X -71.643,Y -29.781,Z -59.270,A -90.000,B 90.000,C 0.000} C_DIS
LIN {X -71.534,Y -29.750,Z -59.149,A -90.000,B 90.000,C 0.000} C_DIS
LIN {X -71.145,Y -29.628,Z -58.723,A -90.000,B 90.000,C 0.000} C_DIS
LIN {X -71.009,Y -29.589,Z -58.583,A -90.000,B 90.000,C 0.000} C_DIS
LIN {X -70.738,Y -29.515,Z -58.318,A -90.000,B 90.000,C 0.000} C_DIS
LIN {X -70.527,Y -29.461,Z -58.124,A -90.000,B 90.000,C 0.000} C_DIS
LIN {X -70.454,Y -29.446,Z -58.058,A -90.000,B 90.000,C 0.000} C_DIS
LIN {X -70.167,Y -29.388,Z -57.815,A -90.000,B 90.000,C 0.000} C_DIS
LIN {X -70.028,Y -29.363,Z -57.706,A -90.000,B 90.000,C 0.000} C_DIS
LIN {X -69.788,Y -29.322,Z -57.528,A -90.000,B 90.000,C 0.000} C_DIS
LIN {X -69.700,Y -29.308,Z -57.466,A -90.000,B 90.000,C 0.000} C_DIS
LIN {X -69.573,Y -29.297,Z -57.374,A -90.000,B 90.000,C 0.000} C_DIS
LIN {X -69.455,Y -29.279,Z -57.284,A -90.000,B 90.000,C 0.000} C_DIS
LIN {X -69.249,Y -29.244,Z -57.114,A -90.000,B 90.000,C 0.000} C_DIS
LIN {X -69.159,Y -29.227,Z -57.033,A -90.000,B 90.000,C 0.000} C_DIS
LIN {X -69.043,Y -29.202,Z -56.918,A -90.000,B 90.000,C 0.000} C_DIS
LIN {X -68.975,Y -29.186,Z -56.845,A -90.000,B 90.000,C 0.000} C_DIS
LIN {X -68.891,Y -29.166,Z -56.741,A -90.000,B 90.000,C 0.000} C_DIS
LIN {X -68.845,Y -29.152,Z -56.676,A -90.000,B 90.000,C 0.000} C_DIS
LIN {X -68.791,Y -29.133,Z -56.584,A -90.000,B 90.000,C 0.000} C_DIS
LIN {X -68.764,Y -29.120,Z -56.526,A -90.000,B 90.000,C 0.000} C_DIS
LIN {X -68.739,Y -29.101,Z -56.446,A -90.000,B 90.000,C 0.000} C_DIS
LIN {X -68.731,Y -29.088,Z -56.396,A -90.000,B 90.000,C 0.000} C_DIS
LIN {X -68.733,Y -29.070,Z -56.327,A -90.000,B 90.000,C 0.000} C_DIS
LIN {X -68.750,Y -29.053,Z -56.265,A -90.000,B 90.000,C 0.000} C_DIS
LIN {X -68.781,Y -29.036,Z -56.211,A -90.000,B 90.000,C 0.000} C_DIS
LIN {X -68.809,Y -29.025,Z -56.178,A -90.000,B 90.000,C 0.000} C_DIS
LIN {X -68.844,Y -29.014,Z -56.149,A -90.000,B 90.000,C 0.000} C_DIS
LIN {X -68.884,Y -29.004,Z -56.123,A -90.000,B 90.000,C 0.000} C_DIS
LIN {X -68.955,Y -28.989,Z -56.090,A -90.000,B 90.000,C 0.000} C_DIS
LIN {X -69.009,Y -28.980,Z -56.072,A -90.000,B 90.000,C 0.000} C_DIS
LIN {X -69.100,Y -28.967,Z -56.051,A -90.000,B 90.000,C 0.000} C_DIS
LIN {X -69.201,Y -28.955,Z -56.038,A -90.000,B 90.000,C 0.000} C_DIS
LIN {X -69.274,Y -28.947,Z -56.033,A -90.000,B 90.000,C 0.000} C_DIS
LIN {X -69.433,Y -28.934,Z -56.034,A -90.000,B 90.000,C 0.000} C_DIS
LIN {X -69.519,Y -28.928,Z -56.039,A -90.000,B 90.000,C 0.000} C_DIS
LIN {X -69.701,Y -28.918,Z -56.059,A -90.000,B 90.000,C 0.000} C_DIS
LIN {X -69.896,Y -28.910,Z -56.093,A -90.000,B 90.000,C 0.000} C_DIS
LIN {X -69.998,Y -28.907,Z -56.115,A -90.000,B 90.000,C 0.000} C_DIS
LIN {X -70.211,Y -28.903,Z -56.169,A -90.000,B 90.000,C 0.000} C_DIS
LIN {X -70.432,Y -28.903,Z -56.237,A -90.000,B 90.000,C 0.000} C_DIS
LIN {X -70.662,Y -28.908,Z -56.319,A -90.000,B 90.000,C 0.000} C_DIS
LIN {X -70.779,Y -28.911,Z -56.365,A -90.000,B 90.000,C 0.000} C_DIS
LIN {X -71.017,Y -28.921,Z -56.468,A -90.000,B 90.000,C 0.000} C_DIS
LIN {X -71.259,Y -28.935,Z -56.585,A -90.000,B 90.000,C 0.000} C_DIS
LIN {X -71.503,Y -28.959,Z -56.716,A -90.000,B 90.000,C 0.000} C_DIS
LIN {X -71.748,Y -28.993,Z -56.861,A -90.000,B 90.000,C 0.000} C_DIS
LIN {X -71.992,Y -29.032,Z -57.020,A -90.000,B 90.000,C 0.000} C_DIS
LIN {X -72.234,Y -29.076,Z -57.194,A -90.000,B 90.000,C 0.000} C_DIS
LIN {X -72.472,Y -29.125,Z -57.383,A -90.000,B 90.000,C 0.000} C_DIS
LIN {X -72.704,Y -29.181,Z -57.586,A -90.000,B 90.000,C 0.000} C_DIS
LIN {X -72.817,Y -29.210,Z -57.693,A -90.000,B 90.000,C 0.000} C_DIS
LIN {X -72.928,Y -29.243,Z -57.804,A -90.000,B 90.000,C 0.000} C_DIS
LIN {X -73.038,Y -29.276,Z -57.918,A -90.000,B 90.000,C 0.000} C_DIS
LIN {X -73.145,Y -29.308,Z -58.036,A -90.000,B 90.000,C 0.000} C_DIS
LIN {X -73.209,Y -29.330,Z -58.110,A -90.000,B 90.000,C 0.000} C_DIS
LIN {X -73.438,Y -29.423,Z -58.367,A -90.000,B 90.000,C 0.000} C_DIS
LIN {X -73.496,Y -29.448,Z -58.436,A -90.000,B 90.000,C 0.000} C_DIS
LIN {X -73.625,Y -29.504,Z -58.592,A -90.000,B 90.000,C 0.000} C_DIS
LIN {X -73.825,Y -29.598,Z -58.851,A -90.000,B 90.000,C 0.000} C_DIS
LIN {X -73.912,Y -29.641,Z -58.969,A -90.000,B 90.000,C 0.000} C_DIS
LIN {X -73.984,Y -29.670,Z -59.071,A -90.000,B 90.000,C 0.000} C_DIS
LIN {X -74.119,Y -29.730,Z -59.277,A -90.000,B 90.000,C 0.000} C_DIS
LIN {X -74.206,Y -29.772,Z -59.410,A -90.000,B 90.000,C 0.000} C_DIS
LIN {X -74.274,Y -29.806,Z -59.518,A -90.000,B 90.000,C 0.000} C_DIS
LIN {X -74.612,Y -29.981,Z -60.091,A -90.000,B 90.000,C 0.000} C_DIS
LIN {X -74.721,Y -30.040,Z -60.283,A -90.000,B 90.000,C 0.000} C_DIS
LIN {X -74.777,Y -30.072,Z -60.389,A -90.000,B 90.000,C 0.000} C_DIS
LIN {X -74.877,Y -30.118,Z -60.592,A -90.000,B 90.000,C 0.000} C_DIS
